Yaskawa INFORM job: A_ROOF_UPPER_0614_2_PAINT_24.JBI

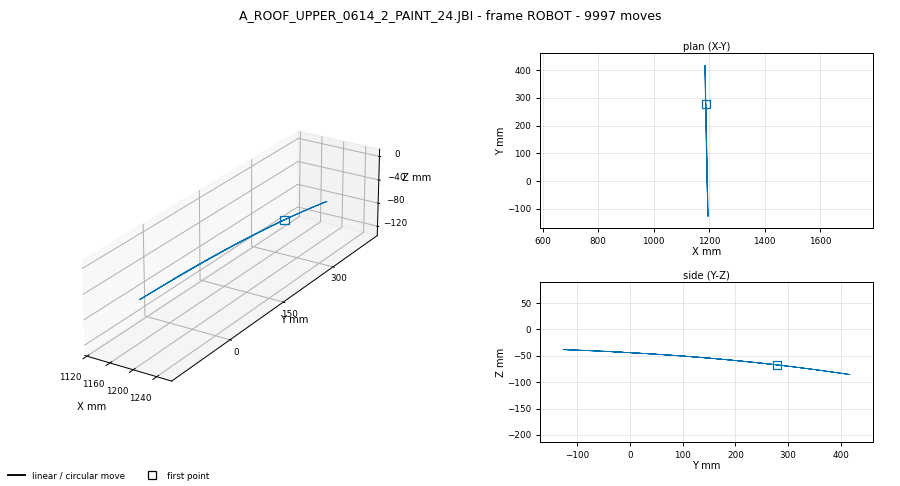
[picture p0: tool path of A_ROOF_UPPER_0614_2_PAINT_24.JBI in frame ROBOT, 9997 of 9997 moves have a stored position in this frame; points joined in program order, loops and branches not executed]
/JOB
//NAME A_ROOF_UPPER_0614_2_PAINT24
//POS
///NPOS 9997,0,0,0,0,0
///TOOL 1
///USER 0
///POSTYPE ROBOT
///RECTAN
///RCONF 1,0,0,0,0,0,0,0,0,0,0,0,0,0,0,0,0,0,0,0,0,0,0,0
C00000=1188.616,279.548,-67.285,-176.910,7.365,148.491
C00001=1188.621,279.299,-67.256,-176.912,7.362,148.491
C00002=1188.625,279.052,-67.228,-176.914,7.359,148.491
C00003=1188.629,278.803,-67.199,-176.917,7.356,148.491
C00004=1188.633,278.555,-67.170,-176.920,7.353,148.491
C00005=1188.638,278.306,-67.142,-176.922,7.351,148.492
C00006=1188.642,278.058,-67.113,-176.925,7.348,148.492
C00007=1188.646,277.809,-67.085,-176.927,7.345,148.492
C00008=1188.651,277.561,-67.056,-176.930,7.343,148.492
C00009=1188.655,277.313,-67.028,-176.932,7.340,148.492
C00010=1188.660,277.065,-67.000,-176.936,7.337,148.492
C00011=1188.664,276.816,-66.971,-176.938,7.335,148.492
C00012=1188.668,276.568,-66.942,-176.940,7.332,148.492
C00013=1188.673,276.320,-66.914,-176.943,7.330,148.492
C00014=1188.677,276.071,-66.885,-176.945,7.327,148.492
C00015=1188.682,275.823,-66.857,-176.948,7.324,148.492
C00016=1188.685,275.574,-66.829,-176.950,7.322,148.492
C00017=1188.690,275.325,-66.800,-176.953,7.319,148.492
C00018=1188.694,275.078,-66.772,-176.956,7.316,148.493
C00019=1188.698,274.829,-66.743,-176.958,7.314,148.493
C00020=1188.703,274.581,-66.715,-176.961,7.311,148.493
C00021=1188.707,274.333,-66.686,-176.964,7.308,148.493
C00022=1188.712,274.085,-66.659,-176.966,7.306,148.493
C00023=1188.716,273.836,-66.630,-176.969,7.303,148.493
C00024=1188.720,273.588,-66.602,-176.971,7.301,148.493
C00025=1188.725,273.339,-66.573,-176.974,7.298,148.493
C00026=1188.729,273.091,-66.546,-176.977,7.295,148.493
C00027=1188.733,272.843,-66.518,-176.979,7.293,148.493
C00028=1188.738,272.594,-66.489,-176.981,7.290,148.493
C00029=1188.742,272.346,-66.461,-176.984,7.287,148.493
C00030=1188.746,272.097,-66.432,-176.986,7.285,148.494
C00031=1188.751,271.849,-66.404,-176.990,7.282,148.494
C00032=1188.755,271.601,-66.377,-176.992,7.280,148.494
C00033=1188.760,271.352,-66.348,-176.994,7.277,148.494
C00034=1188.764,271.104,-66.320,-176.997,7.274,148.494
C00035=1188.768,270.855,-66.291,-176.999,7.272,148.494
C00036=1188.773,270.608,-66.264,-177.002,7.269,148.494
C00037=1188.776,270.359,-66.236,-177.005,7.267,148.494
C00038=1188.782,270.111,-66.207,-177.007,7.264,148.494
C00039=1188.786,269.862,-66.180,-177.010,7.261,148.494
C00040=1188.790,269.614,-66.152,-177.012,7.259,148.495
C00041=1188.794,269.365,-66.123,-177.015,7.256,148.495
C00042=1188.799,269.117,-66.095,-177.018,7.254,148.495
C00043=1188.803,268.868,-66.067,-177.020,7.251,148.495
C00044=1188.808,268.620,-66.039,-177.023,7.248,148.495
C00045=1188.812,268.372,-66.012,-177.025,7.246,148.495
C00046=1188.816,268.123,-65.984,-177.028,7.243,148.495
C00047=1188.821,267.875,-65.955,-177.031,7.241,148.495
C00048=1188.825,267.626,-65.927,-177.033,7.238,148.495
C00049=1188.830,267.378,-65.900,-177.035,7.236,148.496
C00050=1188.834,267.130,-65.872,-177.038,7.233,148.496
C00051=1188.838,266.881,-65.844,-177.041,7.230,148.496
C00052=1188.843,266.633,-65.816,-177.043,7.228,148.496
C00053=1188.847,266.384,-65.788,-177.046,7.225,148.496
C00054=1188.851,266.136,-65.761,-177.048,7.223,148.496
C00055=1188.856,265.888,-65.733,-177.051,7.220,148.496
C00056=1188.860,265.639,-65.705,-177.054,7.218,148.496
C00057=1188.865,265.391,-65.677,-177.056,7.215,148.496
C00058=1188.869,265.143,-65.649,-177.059,7.212,148.497
C00059=1188.873,264.894,-65.622,-177.061,7.210,148.497
C00060=1188.877,264.646,-65.594,-177.064,7.207,148.497
C00061=1188.882,264.396,-65.566,-177.067,7.205,148.497
C00062=1188.887,264.149,-65.538,-177.069,7.202,148.497
C00063=1188.891,263.901,-65.511,-177.072,7.200,148.497
C00064=1188.895,263.652,-65.483,-177.075,7.197,148.497
C00065=1188.899,263.404,-65.455,-177.077,7.194,148.497
C00066=1188.904,263.155,-65.428,-177.080,7.192,148.498
C00067=1188.909,262.882,-65.398,-177.082,7.189,148.498
C00068=1188.914,262.609,-65.367,-177.086,7.186,148.498
C00069=1188.919,262.336,-65.337,-177.088,7.183,148.498
C00070=1188.923,262.064,-65.307,-177.091,7.181,148.498
C00071=1188.928,261.815,-65.280,-177.094,7.179,148.498
C00072=1188.931,261.567,-65.252,-177.096,7.176,148.498
C00073=1188.937,261.318,-65.224,-177.098,7.174,148.498
C00074=1188.941,261.070,-65.196,-177.102,7.171,148.499
C00075=1188.946,260.821,-65.169,-177.104,7.169,148.499
C00076=1188.950,260.573,-65.141,-177.107,7.166,148.499
C00077=1188.954,260.324,-65.114,-177.109,7.164,148.499
C00078=1188.959,260.076,-65.087,-177.112,7.161,148.499
C00079=1188.963,259.827,-65.059,-177.114,7.159,148.499
C00080=1188.967,259.579,-65.032,-177.117,7.156,148.499
C00081=1188.972,259.330,-65.005,-177.120,7.153,148.500
C00082=1188.976,259.082,-64.977,-177.122,7.151,148.500
C00083=1188.980,258.833,-64.949,-177.125,7.148,148.500
C00084=1188.985,258.585,-64.922,-177.128,7.146,148.500
C00085=1188.989,258.337,-64.895,-177.130,7.143,148.500
C00086=1188.994,258.088,-64.868,-177.132,7.141,148.500
C00087=1188.999,257.840,-64.840,-177.135,7.138,148.500
C00088=1189.002,257.592,-64.813,-177.138,7.136,148.500
C00089=1189.006,257.343,-64.786,-177.140,7.133,148.501
C00090=1189.011,257.095,-64.759,-177.143,7.131,148.501
C00091=1189.016,256.846,-64.732,-177.146,7.128,148.501
C00092=1189.020,256.598,-64.705,-177.148,7.126,148.501
C00093=1189.024,256.349,-64.677,-177.151,7.123,148.501
C00094=1189.029,256.100,-64.649,-177.153,7.121,148.501
C00095=1189.033,255.852,-64.622,-177.156,7.118,148.501
C00096=1189.038,255.603,-64.595,-177.158,7.116,148.501
C00097=1189.043,255.355,-64.568,-177.161,7.113,148.502
C00098=1189.046,255.106,-64.541,-177.164,7.111,148.502
C00099=1189.050,254.858,-64.514,-177.166,7.108,148.502
C00100=1189.055,254.610,-64.487,-177.169,7.107,148.502
C00101=1189.060,254.361,-64.460,-177.172,7.104,148.502
C00102=1189.064,254.113,-64.432,-177.174,7.101,148.502
C00103=1189.069,253.864,-64.405,-177.177,7.099,148.503
C00104=1189.073,253.616,-64.379,-177.179,7.097,148.503
C00105=1189.077,253.367,-64.352,-177.182,7.094,148.503
C00106=1189.082,253.118,-64.324,-177.185,7.092,148.503
C00107=1189.086,252.870,-64.297,-177.187,7.089,148.503
C00108=1189.091,252.621,-64.270,-177.189,7.087,148.503
C00109=1189.095,252.373,-64.244,-177.193,7.084,148.504
C00110=1189.100,252.125,-64.217,-177.195,7.082,148.504
C00111=1189.104,251.876,-64.190,-177.197,7.080,148.504
C00112=1189.109,251.628,-64.163,-177.200,7.077,148.504
C00113=1189.113,251.379,-64.136,-177.202,7.075,148.504
C00114=1189.117,251.130,-64.109,-177.206,7.072,148.504
C00115=1189.122,250.882,-64.082,-177.208,7.070,148.504
C00116=1189.126,250.633,-64.055,-177.210,7.067,148.504
C00117=1189.130,250.385,-64.028,-177.213,7.065,148.505
C00118=1189.135,250.137,-64.001,-177.216,7.062,148.505
C00119=1189.140,249.888,-63.975,-177.218,7.060,148.505
C00120=1189.144,249.639,-63.948,-177.221,7.057,148.505
C00121=1189.148,249.391,-63.921,-177.223,7.055,148.505
C00122=1189.153,249.142,-63.894,-177.227,7.053,148.506
C00123=1189.157,248.894,-63.868,-177.229,7.050,148.506
C00124=1189.162,248.646,-63.841,-177.231,7.048,148.506
C00125=1189.166,248.397,-63.814,-177.234,7.046,148.506
C00126=1189.170,248.148,-63.788,-177.236,7.043,148.506
C00127=1189.175,247.900,-63.761,-177.239,7.041,148.506
C00128=1189.180,247.651,-63.734,-177.242,7.039,148.507
C00129=1189.184,247.403,-63.707,-177.245,7.036,148.507
C00130=1189.189,247.154,-63.681,-177.247,7.034,148.507
C00131=1189.193,246.906,-63.654,-177.250,7.031,148.507
C00132=1189.197,246.657,-63.627,-177.252,7.029,148.507
C00133=1189.202,246.409,-63.600,-177.255,7.027,148.507
C00134=1189.206,246.160,-63.575,-177.258,7.024,148.508
C00135=1189.211,245.912,-63.548,-177.260,7.022,148.508
C00136=1189.215,245.663,-63.521,-177.263,7.019,148.508
C00137=1189.220,245.414,-63.495,-177.265,7.017,148.508
C00138=1189.224,245.166,-63.468,-177.268,7.014,148.508
C00139=1189.228,244.918,-63.441,-177.271,7.012,148.509
C00140=1189.232,244.669,-63.415,-177.273,7.010,148.509
C00141=1189.237,244.420,-63.388,-177.276,7.008,148.509
C00142=1189.241,244.171,-63.363,-177.278,7.005,148.509
C00143=1189.246,243.923,-63.336,-177.281,7.002,148.509
C00144=1189.250,243.675,-63.309,-177.284,7.001,148.509
C00145=1189.255,243.426,-63.283,-177.286,6.998,148.509
C00146=1189.259,243.178,-63.256,-177.289,6.996,148.510
C00147=1189.264,242.928,-63.230,-177.291,6.994,148.510
C00148=1189.268,242.680,-63.203,-177.294,6.991,148.510
C00149=1189.273,242.431,-63.177,-177.296,6.989,148.510
C00150=1189.277,242.184,-63.151,-177.299,6.987,148.511
C00151=1189.282,241.935,-63.125,-177.302,6.984,148.511
C00152=1189.286,241.686,-63.098,-177.304,6.982,148.511
C00153=1189.291,241.437,-63.072,-177.307,6.979,148.511
C00154=1189.295,241.189,-63.045,-177.310,6.977,148.511
C00155=1189.299,240.940,-63.020,-177.312,6.975,148.511
C00156=1189.304,240.692,-62.993,-177.315,6.972,148.511
C00157=1189.308,240.443,-62.967,-177.317,6.970,148.512
C00158=1189.313,240.194,-62.941,-177.320,6.967,148.512
C00159=1189.317,239.946,-62.914,-177.323,6.966,148.512
C00160=1189.322,239.698,-62.889,-177.325,6.963,148.512
C00161=1189.326,239.449,-62.862,-177.328,6.961,148.513
C00162=1189.331,239.200,-62.836,-177.330,6.959,148.513
C00163=1189.335,238.951,-62.810,-177.333,6.956,148.513
C00164=1189.339,238.703,-62.783,-177.336,6.954,148.513
C00165=1189.344,238.454,-62.757,-177.338,6.952,148.513
C00166=1189.348,238.206,-62.732,-177.341,6.949,148.513
C00167=1189.353,237.958,-62.705,-177.344,6.947,148.514
C00168=1189.357,237.709,-62.679,-177.346,6.945,148.514
C00169=1189.362,237.460,-62.653,-177.349,6.942,148.514
C00170=1189.367,237.211,-62.627,-177.351,6.940,148.514
C00171=1189.372,236.940,-62.599,-177.354,6.938,148.515
C00172=1189.376,236.668,-62.571,-177.358,6.935,148.515
C00173=1189.381,236.397,-62.542,-177.360,6.933,148.515
C00174=1189.385,236.125,-62.514,-177.363,6.930,148.515
C00175=1189.391,235.877,-62.488,-177.366,6.928,148.516
C00176=1189.395,235.629,-62.461,-177.368,6.925,148.516
C00177=1189.399,235.380,-62.436,-177.371,6.923,148.516
C00178=1189.403,235.131,-62.410,-177.373,6.921,148.516
C00179=1189.408,234.882,-62.383,-177.376,6.919,148.516
C00180=1189.413,234.634,-62.358,-177.379,6.916,148.516
C00181=1189.417,234.385,-62.332,-177.381,6.915,148.517
C00182=1189.421,234.136,-62.307,-177.384,6.912,148.517
C00183=1189.425,233.888,-62.280,-177.387,6.910,148.517
C00184=1189.431,233.639,-62.254,-177.389,6.908,148.517
C00185=1189.435,233.391,-62.228,-177.392,6.905,148.518
C00186=1189.439,233.142,-62.203,-177.394,6.903,148.518
C00187=1189.444,232.893,-62.177,-177.397,6.901,148.518
C00188=1189.448,232.645,-62.151,-177.400,6.898,148.518
C00189=1189.453,232.396,-62.126,-177.402,6.896,148.518
C00190=1189.457,232.147,-62.100,-177.405,6.894,148.519
C00191=1189.462,231.899,-62.074,-177.407,6.891,148.519
C00192=1189.467,231.650,-62.048,-177.410,6.890,148.519
C00193=1189.471,231.401,-62.023,-177.412,6.887,148.519
C00194=1189.475,231.153,-61.997,-177.416,6.885,148.519
C00195=1189.480,230.904,-61.971,-177.418,6.883,148.520
C00196=1189.484,230.656,-61.946,-177.420,6.881,148.520
C00197=1189.488,230.407,-61.920,-177.424,6.878,148.520
C00198=1189.493,230.159,-61.894,-177.426,6.876,148.520
C00199=1189.497,229.910,-61.869,-177.428,6.874,148.521
C00200=1189.502,229.661,-61.843,-177.431,6.871,148.521
C00201=1189.507,229.412,-61.818,-177.434,6.869,148.521
C00202=1189.511,229.164,-61.793,-177.436,6.868,148.521
C00203=1189.515,228.915,-61.767,-177.439,6.865,148.521
C00204=1189.520,228.667,-61.741,-177.442,6.863,148.522
C00205=1189.524,228.418,-61.716,-177.444,6.861,148.522
C00206=1189.529,228.169,-61.690,-177.447,6.858,148.522
C00207=1189.533,227.921,-61.665,-177.450,6.856,148.522
C00208=1189.538,227.672,-61.640,-177.452,6.854,148.523
C00209=1189.543,227.423,-61.614,-177.455,6.852,148.523
C00210=1189.547,227.175,-61.588,-177.457,6.849,148.523
C00211=1189.551,226.926,-61.563,-177.460,6.847,148.523
C00212=1189.556,226.678,-61.537,-177.463,6.846,148.524
C00213=1189.561,226.428,-61.512,-177.465,6.843,148.524
C00214=1189.565,226.179,-61.486,-177.468,6.841,148.524
C00215=1189.570,225.931,-61.461,-177.471,6.839,148.524
C00216=1189.574,225.682,-61.436,-177.473,6.836,148.524
C00217=1189.579,225.434,-61.411,-177.476,6.834,148.525
C00218=1189.583,225.185,-61.385,-177.478,6.832,148.525
C00219=1189.588,224.937,-61.360,-177.481,6.830,148.525
C00220=1189.593,224.688,-61.334,-177.484,6.828,148.526
C00221=1189.597,224.439,-61.309,-177.486,6.825,148.526
C00222=1189.602,224.190,-61.284,-177.489,6.824,148.526
C00223=1189.605,223.941,-61.259,-177.492,6.821,148.526
C00224=1189.610,223.693,-61.234,-177.494,6.819,148.526
C00225=1189.615,223.444,-61.208,-177.497,6.817,148.527
C00226=1189.620,223.196,-61.183,-177.500,6.815,148.527
C00227=1189.624,222.947,-61.157,-177.502,6.812,148.527
C00228=1189.629,222.698,-61.133,-177.505,6.810,148.527
C00229=1189.632,222.450,-61.108,-177.507,6.808,148.528
C00230=1189.638,222.201,-61.083,-177.510,6.806,148.528
C00231=1189.642,221.952,-61.057,-177.513,6.804,148.528
C00232=1189.646,221.703,-61.032,-177.515,6.802,148.528
C00233=1189.651,221.455,-61.007,-177.518,6.800,148.529
C00234=1189.655,221.206,-60.982,-177.521,6.797,148.529
C00235=1189.660,220.958,-60.957,-177.523,6.795,148.529
C00236=1189.664,220.708,-60.932,-177.526,6.793,148.529
C00237=1189.669,220.460,-60.906,-177.529,6.791,148.530
C00238=1189.674,220.211,-60.881,-177.531,6.788,148.530
C00239=1189.678,219.963,-60.857,-177.534,6.787,148.530
C00240=1189.682,219.713,-60.832,-177.537,6.785,148.530
C00241=1189.687,219.465,-60.806,-177.539,6.783,148.531
C00242=1189.691,219.217,-60.782,-177.542,6.780,148.531
C00243=1189.696,218.967,-60.757,-177.545,6.778,148.531
C00244=1189.701,218.719,-60.732,-177.547,6.776,148.532
C00245=1189.705,218.470,-60.707,-177.549,6.774,148.532
C00246=1189.709,218.222,-60.682,-177.553,6.772,148.532
C00247=1189.714,217.973,-60.657,-177.555,6.770,148.532
C00248=1189.719,217.724,-60.632,-177.557,6.768,148.532
C00249=1189.723,217.475,-60.607,-177.560,6.766,148.533
C00250=1189.728,217.227,-60.582,-177.563,6.763,148.533
C00251=1189.733,216.978,-60.558,-177.565,6.761,148.533
C00252=1189.737,216.729,-60.533,-177.568,6.759,148.533
C00253=1189.741,216.481,-60.508,-177.571,6.757,148.534
C00254=1189.745,216.232,-60.483,-177.574,6.755,148.534
C00255=1189.750,215.983,-60.459,-177.576,6.753,148.534
C00256=1189.755,215.734,-60.433,-177.579,6.751,148.535
C00257=1189.759,215.486,-60.409,-177.581,6.749,148.535
C00258=1189.764,215.237,-60.384,-177.584,6.747,148.535
C00259=1189.769,214.988,-60.359,-177.587,6.744,148.535
C00260=1189.773,214.739,-60.335,-177.590,6.742,148.536
C00261=1189.778,214.491,-60.310,-177.592,6.741,148.536
C00262=1189.782,214.242,-60.285,-177.594,6.738,148.536
C00263=1189.787,213.993,-60.261,-177.598,6.736,148.536
C00264=1189.791,213.744,-60.236,-177.600,6.734,148.537
C00265=1189.796,213.495,-60.212,-177.603,6.732,148.537
C00266=1189.800,213.247,-60.187,-177.605,6.730,148.537
C00267=1189.804,212.998,-60.162,-177.608,6.727,148.537
C00268=1189.809,212.750,-60.138,-177.611,6.726,148.538
C00269=1189.814,212.501,-60.113,-177.613,6.723,148.538
C00270=1189.818,212.252,-60.088,-177.616,6.722,148.538
C00271=1189.823,212.003,-60.064,-177.618,6.720,148.539
C00272=1189.828,211.755,-60.039,-177.622,6.717,148.539
C00273=1189.832,211.505,-60.015,-177.624,6.715,148.539
C00274=1189.836,211.257,-59.991,-177.626,6.713,148.539
C00275=1189.841,210.987,-59.964,-177.629,6.711,148.540
C00276=1189.846,210.717,-59.937,-177.632,6.709,148.540
C00277=1189.851,210.446,-59.910,-177.635,6.707,148.540
C00278=1189.856,210.175,-59.884,-177.638,6.704,148.541
C00279=1189.861,209.927,-59.860,-177.641,6.703,148.541
C00280=1189.865,209.677,-59.835,-177.643,6.700,148.541
C00281=1189.870,209.429,-59.811,-177.646,6.699,148.541
C00282=1189.875,209.180,-59.786,-177.649,6.696,148.542
C00283=1189.879,208.932,-59.762,-177.652,6.694,148.542
C00284=1189.883,208.682,-59.738,-177.654,6.692,148.542
C00285=1189.888,208.434,-59.713,-177.656,6.690,148.543
C00286=1189.893,208.185,-59.689,-177.659,6.688,148.543
C00287=1189.898,207.937,-59.664,-177.662,6.686,148.543
C00288=1189.902,207.688,-59.640,-177.664,6.684,148.543
C00289=1189.906,207.438,-59.617,-177.667,6.682,148.544
C00290=1189.911,207.190,-59.592,-177.670,6.680,148.544
C00291=1189.916,206.941,-59.568,-177.672,6.678,148.544
C00292=1189.920,206.692,-59.543,-177.676,6.676,148.545
C00293=1189.925,206.444,-59.519,-177.678,6.673,148.545
C00294=1189.929,206.195,-59.495,-177.681,6.672,148.545
C00295=1189.934,205.946,-59.471,-177.683,6.670,148.545
C00296=1189.939,205.697,-59.447,-177.686,6.668,148.546
C00297=1189.943,205.448,-59.422,-177.688,6.666,148.546
C00298=1189.947,205.200,-59.398,-177.691,6.663,148.546
C00299=1189.953,204.950,-59.374,-177.694,6.661,148.547
C00300=1189.957,204.702,-59.350,-177.697,6.660,148.547
C00301=1189.961,204.454,-59.326,-177.699,6.658,148.547
C00302=1189.965,204.205,-59.302,-177.702,6.656,148.548
C00303=1189.971,203.955,-59.278,-177.704,6.654,148.548
C00304=1189.975,203.707,-59.254,-177.707,6.652,148.548
C00305=1189.979,203.458,-59.229,-177.710,6.649,148.548
C00306=1189.984,203.209,-59.206,-177.713,6.648,148.549
C00307=1189.989,202.961,-59.181,-177.715,6.646,148.549
C00308=1189.993,202.712,-59.157,-177.717,6.644,148.549
C00309=1189.998,202.462,-59.134,-177.720,6.642,148.550
C00310=1190.002,202.214,-59.110,-177.723,6.640,148.550
C00311=1190.006,201.966,-59.085,-177.725,6.638,148.550
C00312=1190.011,201.717,-59.062,-177.729,6.636,148.551
C00313=1190.016,201.468,-59.037,-177.731,6.633,148.551
C00314=1190.021,201.219,-59.014,-177.733,6.632,148.551
C00315=1190.025,200.970,-58.990,-177.736,6.630,148.551
C00316=1190.029,200.721,-58.966,-177.739,6.628,148.552
C00317=1190.034,200.472,-58.942,-177.741,6.626,148.552
C00318=1190.038,200.224,-58.918,-177.744,6.624,148.552
C00319=1190.044,199.975,-58.894,-177.747,6.621,148.553
C00320=1190.048,199.726,-58.870,-177.749,6.620,148.553
C00321=1190.053,199.477,-58.847,-177.752,6.618,148.553
C00322=1190.057,199.229,-58.823,-177.755,6.616,148.554
C00323=1190.062,198.980,-58.799,-177.757,6.614,148.554
C00324=1190.067,198.731,-58.776,-177.760,6.612,148.554
C00325=1190.071,198.482,-58.752,-177.762,6.610,148.554
C00326=1190.076,198.233,-58.729,-177.765,6.608,148.555
C00327=1190.079,197.984,-58.704,-177.768,6.606,148.555
C00328=1190.084,197.735,-58.681,-177.771,6.604,148.555
C00329=1190.089,197.487,-58.657,-177.774,6.602,148.556
C00330=1190.093,197.238,-58.633,-177.776,6.600,148.556
C00331=1190.098,196.989,-58.610,-177.778,6.598,148.556
C00332=1190.103,196.740,-58.585,-177.781,6.597,148.557
C00333=1190.108,196.491,-58.562,-177.784,6.595,148.557
C00334=1190.113,196.242,-58.539,-177.786,6.593,148.557
C00335=1190.117,195.993,-58.514,-177.789,6.591,148.558
C00336=1190.122,195.744,-58.491,-177.792,6.589,148.558
C00337=1190.126,195.495,-58.468,-177.795,6.587,148.558
C00338=1190.131,195.247,-58.444,-177.797,6.585,148.558
C00339=1190.135,194.998,-58.420,-177.800,6.583,148.559
C00340=1190.140,194.749,-58.397,-177.802,6.581,148.559
C00341=1190.144,194.501,-58.373,-177.805,6.579,148.559
C00342=1190.148,194.252,-58.350,-177.808,6.577,148.560
C00343=1190.153,194.003,-58.327,-177.810,6.576,148.560
C00344=1190.158,193.754,-58.303,-177.813,6.574,148.560
C00345=1190.162,193.505,-58.279,-177.816,6.572,148.561
C00346=1190.167,193.256,-58.256,-177.818,6.570,148.561
C00347=1190.172,193.007,-58.233,-177.821,6.568,148.561
C00348=1190.176,192.758,-58.209,-177.824,6.565,148.562
C00349=1190.181,192.509,-58.186,-177.826,6.564,148.562
C00350=1190.185,192.261,-58.162,-177.829,6.562,148.562
C00351=1190.191,192.012,-58.139,-177.832,6.560,148.563
C00352=1190.195,191.763,-58.115,-177.834,6.558,148.563
C00353=1190.199,191.515,-58.093,-177.837,6.556,148.563
C00354=1190.204,191.266,-58.069,-177.840,6.555,148.564
C00355=1190.209,191.017,-58.046,-177.842,6.552,148.564
C00356=1190.213,190.767,-58.023,-177.845,6.551,148.564
C00357=1190.218,190.518,-57.999,-177.847,6.549,148.565
C00358=1190.223,190.269,-57.976,-177.850,6.547,148.565
C00359=1190.227,190.021,-57.952,-177.853,6.545,148.565
C00360=1190.231,189.772,-57.929,-177.855,6.543,148.566
C00361=1190.236,189.523,-57.906,-177.858,6.542,148.566
C00362=1190.241,189.274,-57.882,-177.861,6.540,148.566
C00363=1190.246,189.026,-57.859,-177.864,6.537,148.567
C00364=1190.251,188.777,-57.836,-177.866,6.535,148.567
C00365=1190.255,188.528,-57.813,-177.869,6.533,148.567
C00366=1190.259,188.279,-57.790,-177.871,6.531,148.568
C00367=1190.264,188.030,-57.767,-177.874,6.530,148.568
C00368=1190.269,187.781,-57.743,-177.877,6.528,148.568
C00369=1190.273,187.532,-57.720,-177.879,6.526,148.569
C00370=1190.277,187.283,-57.697,-177.882,6.524,148.569
C00371=1190.283,187.034,-57.675,-177.885,6.523,148.569
C00372=1190.288,186.785,-57.651,-177.887,6.521,148.570
C00373=1190.292,186.537,-57.629,-177.890,6.519,148.570
C00374=1190.296,186.288,-57.605,-177.893,6.517,148.570
C00375=1190.301,186.039,-57.582,-177.895,6.515,148.571
C00376=1190.306,185.789,-57.559,-177.898,6.514,148.571
C00377=1190.310,185.541,-57.536,-177.901,6.512,148.571
C00378=1190.315,185.292,-57.513,-177.903,6.510,148.572
C00379=1190.320,185.023,-57.488,-177.906,6.508,148.572
C00380=1190.325,184.753,-57.463,-177.909,6.506,148.572
C00381=1190.330,184.483,-57.438,-177.912,6.504,148.573
C00382=1190.335,184.214,-57.414,-177.915,6.502,148.573
C00383=1190.340,183.965,-57.391,-177.917,6.500,148.574
C00384=1190.344,183.716,-57.367,-177.920,6.498,148.574
C00385=1190.348,183.467,-57.345,-177.923,6.497,148.574
C00386=1190.354,183.218,-57.322,-177.925,6.495,148.575
C00387=1190.358,182.969,-57.299,-177.928,6.493,148.575
C00388=1190.362,182.721,-57.276,-177.931,6.491,148.575
C00389=1190.367,182.471,-57.253,-177.933,6.489,148.576
C00390=1190.371,182.222,-57.231,-177.935,6.487,148.576
C00391=1190.377,181.974,-57.208,-177.938,6.485,148.576
C00392=1190.381,181.725,-57.185,-177.941,6.484,148.576
C00393=1190.386,181.475,-57.162,-177.943,6.482,148.577
C00394=1190.390,181.226,-57.139,-177.946,6.480,148.577
C00395=1190.395,180.978,-57.116,-177.949,6.478,148.578
C00396=1190.400,180.729,-57.094,-177.951,6.476,148.578
C00397=1190.404,180.480,-57.071,-177.954,6.475,148.578
C00398=1190.409,180.232,-57.048,-177.957,6.473,148.579
C00399=1190.413,179.982,-57.026,-177.959,6.471,148.579
C00400=1190.418,179.733,-57.003,-177.962,6.469,148.579
C00401=1190.422,179.484,-56.981,-177.965,6.468,148.580
C00402=1190.428,179.236,-56.958,-177.967,6.466,148.580
C00403=1190.432,178.987,-56.935,-177.970,6.464,148.580
C00404=1190.437,178.737,-56.912,-177.973,6.462,148.581
C00405=1190.441,178.489,-56.890,-177.975,6.460,148.581
C00406=1190.446,178.240,-56.867,-177.978,6.459,148.582
C00407=1190.450,177.991,-56.844,-177.981,6.457,148.582
C00408=1190.456,177.742,-56.822,-177.983,6.455,148.582
C00409=1190.460,177.493,-56.799,-177.986,6.453,148.583
C00410=1190.465,177.244,-56.777,-177.989,6.451,148.583
C00411=1190.469,176.995,-56.754,-177.991,6.450,148.583
C00412=1190.474,176.746,-56.732,-177.994,6.448,148.584
C00413=1190.478,176.497,-56.709,-177.997,6.446,148.584
C00414=1190.483,176.248,-56.687,-177.999,6.444,148.584
C00415=1190.488,175.999,-56.664,-178.002,6.442,148.585
C00416=1190.492,175.750,-56.642,-178.005,6.441,148.585
C00417=1190.497,175.501,-56.620,-178.008,6.439,148.585
C00418=1190.502,175.252,-56.597,-178.010,6.437,148.586
C00419=1190.506,175.003,-56.575,-178.013,6.435,148.586
C00420=1190.511,174.755,-56.552,-178.016,6.434,148.587
C00421=1190.516,174.505,-56.530,-178.018,6.432,148.587
C00422=1190.520,174.256,-56.508,-178.021,6.430,148.587
C00423=1190.525,174.008,-56.485,-178.024,6.428,148.588
C00424=1190.529,173.758,-56.463,-178.026,6.426,148.588
C00425=1190.534,173.510,-56.441,-178.028,6.425,148.588
C00426=1190.539,173.261,-56.418,-178.031,6.424,148.589
C00427=1190.543,173.011,-56.395,-178.034,6.422,148.589
C00428=1190.548,172.763,-56.374,-178.036,6.420,148.589
C00429=1190.553,172.514,-56.350,-178.039,6.418,148.590
C00430=1190.558,172.265,-56.329,-178.042,6.416,148.590
C00431=1190.562,172.016,-56.307,-178.044,6.415,148.591
C00432=1190.568,171.767,-56.284,-178.047,6.413,148.591
C00433=1190.572,171.518,-56.262,-178.050,6.411,148.591
C00434=1190.576,171.269,-56.240,-178.052,6.409,148.592
C00435=1190.581,171.020,-56.218,-178.055,6.408,148.592
C00436=1190.586,170.770,-56.195,-178.058,6.406,148.592
C00437=1190.590,170.522,-56.173,-178.060,6.404,148.593
C00438=1190.595,170.273,-56.151,-178.063,6.402,148.593
C00439=1190.599,170.024,-56.129,-178.066,6.400,148.593
C00440=1190.604,169.775,-56.107,-178.068,6.399,148.594
C00441=1190.609,169.526,-56.085,-178.071,6.398,148.594
C00442=1190.614,169.277,-56.063,-178.074,6.396,148.595
C00443=1190.618,169.029,-56.040,-178.076,6.394,148.595
C00444=1190.622,168.779,-56.018,-178.079,6.393,148.596
C00445=1190.628,168.531,-55.996,-178.082,6.391,148.596
C00446=1190.632,168.281,-55.974,-178.084,6.389,148.596
C00447=1190.637,168.033,-55.952,-178.087,6.387,148.597
C00448=1190.641,167.783,-55.930,-178.090,6.385,148.597
C00449=1190.646,167.535,-55.909,-178.092,6.384,148.597
C00450=1190.651,167.285,-55.886,-178.095,6.382,148.598
C00451=1190.656,167.036,-55.864,-178.097,6.381,148.598
C00452=1190.660,166.787,-55.842,-178.100,6.379,148.599
C00453=1190.665,166.538,-55.821,-178.103,6.377,148.599
C00454=1190.670,166.289,-55.798,-178.105,6.376,148.599
C00455=1190.674,166.040,-55.777,-178.108,6.374,148.600
C00456=1190.679,165.791,-55.755,-178.111,6.372,148.600
C00457=1190.684,165.542,-55.733,-178.113,6.370,148.600
C00458=1190.688,165.294,-55.711,-178.116,6.368,148.601
C00459=1190.693,165.044,-55.689,-178.119,6.367,148.601
C00460=1190.698,164.795,-55.667,-178.122,6.365,148.602
C00461=1190.703,164.546,-55.645,-178.124,6.364,148.602
C00462=1190.707,164.297,-55.623,-178.127,6.362,148.602
C00463=1190.712,164.048,-55.601,-178.129,6.361,148.603
C00464=1190.717,163.799,-55.580,-178.132,6.359,148.603
C00465=1190.721,163.550,-55.558,-178.135,6.357,148.604
C00466=1190.726,163.301,-55.536,-178.137,6.355,148.604
C00467=1190.731,163.053,-55.514,-178.140,6.354,148.604
C00468=1190.735,162.803,-55.492,-178.143,6.352,148.605
C00469=1190.740,162.554,-55.471,-178.145,6.351,148.605
C00470=1190.744,162.305,-55.449,-178.147,6.349,148.605
C00471=1190.749,162.056,-55.427,-178.151,6.348,148.606
C00472=1190.754,161.808,-55.406,-178.153,6.346,148.606
C00473=1190.758,161.558,-55.384,-178.156,6.344,148.607
C00474=1190.763,161.310,-55.362,-178.159,6.342,148.607
C00475=1190.768,161.060,-55.341,-178.161,6.341,148.607
C00476=1190.773,160.811,-55.319,-178.163,6.340,148.608
C00477=1190.777,160.562,-55.297,-178.166,6.338,148.608
C00478=1190.782,160.313,-55.275,-178.169,6.336,148.609
C00479=1190.787,160.064,-55.254,-178.171,6.334,148.609
C00480=1190.792,159.815,-55.233,-178.174,6.332,148.609
C00481=1190.795,159.566,-55.211,-178.177,6.331,148.610
C00482=1190.800,159.317,-55.190,-178.180,6.329,148.610
C00483=1190.806,159.048,-55.166,-178.183,6.327,148.611
C00484=1190.810,158.779,-55.143,-178.185,6.326,148.611
C00485=1190.816,158.510,-55.119,-178.188,6.324,148.612
C00486=1190.820,158.241,-55.097,-178.191,6.322,148.612
C00487=1190.825,157.992,-55.076,-178.194,6.321,148.612
C00488=1190.830,157.743,-55.054,-178.196,6.319,148.613
C00489=1190.835,157.494,-55.032,-178.199,6.318,148.613
C00490=1190.840,157.245,-55.011,-178.201,6.316,148.614
C00491=1190.845,156.996,-54.989,-178.204,6.314,148.614
C00492=1190.850,156.747,-54.968,-178.207,6.313,148.615
C00493=1190.853,156.498,-54.947,-178.210,6.311,148.615
C00494=1190.858,156.249,-54.925,-178.212,6.309,148.615
C00495=1190.863,156.000,-54.904,-178.215,6.308,148.616
C00496=1190.868,155.751,-54.882,-178.217,6.307,148.616
C00497=1190.873,155.502,-54.860,-178.220,6.305,148.616
C00498=1190.878,155.253,-54.839,-178.223,6.303,148.617
C00499=1190.882,155.004,-54.818,-178.226,6.302,148.617
C00500=1190.886,154.754,-54.797,-178.228,6.300,148.618
C00501=1190.891,154.506,-54.775,-178.231,6.299,148.618
C00502=1190.896,154.256,-54.754,-178.233,6.297,148.619
C00503=1190.901,154.008,-54.733,-178.236,6.295,148.619
C00504=1190.905,153.758,-54.712,-178.239,6.294,148.619
C00505=1190.910,153.510,-54.690,-178.241,6.292,148.620
C00506=1190.915,153.260,-54.669,-178.244,6.291,148.620
C00507=1190.920,153.011,-54.649,-178.247,6.289,148.621
C00508=1190.925,152.763,-54.627,-178.249,6.288,148.621
C00509=1190.929,152.513,-54.606,-178.252,6.286,148.621
C00510=1190.934,152.264,-54.584,-178.255,6.284,148.622
C00511=1190.938,152.015,-54.564,-178.257,6.283,148.622
C00512=1190.943,151.767,-54.542,-178.260,6.282,148.623
C00513=1190.948,151.517,-54.521,-178.263,6.280,148.623
C00514=1190.952,151.268,-54.500,-178.265,6.278,148.624
C00515=1190.957,151.019,-54.479,-178.268,6.276,148.624
C00516=1190.962,150.770,-54.458,-178.270,6.275,148.624
C00517=1190.968,150.520,-54.437,-178.273,6.274,148.625
C00518=1190.972,150.272,-54.416,-178.276,6.272,148.625
C00519=1190.976,150.022,-54.394,-178.279,6.271,148.626
C00520=1190.981,149.773,-54.374,-178.281,6.269,148.626
C00521=1190.986,149.525,-54.352,-178.283,6.268,148.626
C00522=1190.991,149.275,-54.331,-178.286,6.266,148.627
C00523=1190.995,149.026,-54.311,-178.289,6.264,148.627
C00524=1191.000,148.778,-54.289,-178.292,6.263,148.628
C00525=1191.005,148.528,-54.268,-178.295,6.261,148.628
C00526=1191.009,148.279,-54.248,-178.297,6.260,148.629
C00527=1191.014,148.030,-54.227,-178.299,6.258,148.629
C00528=1191.018,147.781,-54.206,-178.302,6.257,148.629
C00529=1191.023,147.532,-54.185,-178.305,6.255,148.630
C00530=1191.029,147.283,-54.164,-178.307,6.254,148.630
C00531=1191.033,147.034,-54.143,-178.310,6.252,148.631
C00532=1191.038,146.784,-54.122,-178.313,6.251,148.631
C00533=1191.042,146.536,-54.101,-178.315,6.249,148.631
C00534=1191.048,146.287,-54.080,-178.318,6.248,148.632
C00535=1191.051,146.037,-54.060,-178.321,6.246,148.632
C00536=1191.057,145.788,-54.039,-178.323,6.245,148.633
C00537=1191.061,145.539,-54.018,-178.326,6.243,148.633
C00538=1191.066,145.290,-53.997,-178.328,6.242,148.634
C00539=1191.071,145.041,-53.977,-178.331,6.240,148.634
C00540=1191.076,144.792,-53.956,-178.334,6.239,148.635
C00541=1191.080,144.543,-53.935,-178.337,6.237,148.635
C00542=1191.085,144.294,-53.914,-178.339,6.236,148.635
C00543=1191.090,144.045,-53.893,-178.342,6.234,148.636
C00544=1191.095,143.796,-53.872,-178.344,6.233,148.636
C00545=1191.099,143.547,-53.852,-178.347,6.231,148.637
C00546=1191.104,143.298,-53.831,-178.350,6.230,148.637
C00547=1191.109,143.049,-53.811,-178.352,6.228,148.638
C00548=1191.114,142.799,-53.790,-178.355,6.227,148.638
C00549=1191.118,142.550,-53.769,-178.358,6.225,148.639
C00550=1191.122,142.301,-53.749,-178.360,6.224,148.639
C00551=1191.127,142.051,-53.728,-178.363,6.222,148.639
C00552=1191.132,141.803,-53.707,-178.366,6.221,148.640
C00553=1191.137,141.553,-53.686,-178.368,6.219,148.640
C00554=1191.141,141.304,-53.666,-178.371,6.218,148.641
C00555=1191.146,141.055,-53.646,-178.374,6.217,148.641
C00556=1191.151,140.806,-53.625,-178.376,6.215,148.642
C00557=1191.156,140.557,-53.604,-178.379,6.213,148.642
C00558=1191.161,140.308,-53.583,-178.381,6.212,148.643
C00559=1191.165,140.059,-53.563,-178.384,6.211,148.643
C00560=1191.170,139.809,-53.543,-178.387,6.209,148.643
C00561=1191.175,139.560,-53.522,-178.389,6.208,148.644
C00562=1191.179,139.311,-53.502,-178.392,6.207,148.644
C00563=1191.184,139.062,-53.482,-178.395,6.205,148.645
C00564=1191.189,138.813,-53.461,-178.398,6.203,148.645
C00565=1191.194,138.565,-53.441,-178.400,6.202,148.645
C00566=1191.199,138.316,-53.420,-178.403,6.201,148.646
C00567=1191.204,138.066,-53.400,-178.406,6.199,148.646
C00568=1191.208,137.817,-53.380,-178.408,6.198,148.647
C00569=1191.213,137.568,-53.359,-178.410,6.196,148.647
C00570=1191.218,137.319,-53.338,-178.413,6.195,148.648
C00571=1191.223,137.070,-53.318,-178.416,6.193,148.648
C00572=1191.227,136.820,-53.298,-178.418,6.192,148.649
C00573=1191.232,136.571,-53.278,-178.421,6.190,148.649
C00574=1191.237,136.322,-53.257,-178.424,6.189,148.650
C00575=1191.241,136.073,-53.237,-178.426,6.188,148.650
C00576=1191.246,135.823,-53.217,-178.429,6.186,148.650
C00577=1191.251,135.575,-53.197,-178.432,6.184,148.651
C00578=1191.256,135.325,-53.176,-178.434,6.184,148.651
C00579=1191.261,135.077,-53.156,-178.437,6.182,148.652
C00580=1191.265,134.827,-53.136,-178.440,6.180,148.652
C00581=1191.270,134.579,-53.116,-178.442,6.179,148.653
C00582=1191.275,134.329,-53.095,-178.445,6.178,148.653
C00583=1191.280,134.080,-53.075,-178.448,6.176,148.654
C00584=1191.284,133.831,-53.055,-178.450,6.175,148.654
C00585=1191.289,133.582,-53.034,-178.452,6.173,148.654
C00586=1191.293,133.332,-53.015,-178.456,6.172,148.655
C00587=1191.299,133.064,-52.992,-178.458,6.170,148.655
C00588=1191.304,132.795,-52.971,-178.461,6.169,148.656
C00589=1191.309,132.526,-52.949,-178.464,6.168,148.656
C00590=1191.314,132.258,-52.928,-178.467,6.167,148.657
C00591=1191.319,132.008,-52.907,-178.469,6.165,148.657
C00592=1191.324,131.759,-52.887,-178.472,6.163,148.658
C00593=1191.329,131.511,-52.868,-178.474,6.162,148.658
C00594=1191.334,131.262,-52.847,-178.477,6.161,148.659
C00595=1191.338,131.013,-52.827,-178.480,6.159,148.659
C00596=1191.343,130.763,-52.807,-178.482,6.158,148.660
C00597=1191.347,130.514,-52.787,-178.485,6.157,148.660
C00598=1191.353,130.265,-52.768,-178.488,6.155,148.661
C00599=1191.357,130.016,-52.747,-178.490,6.154,148.661
C00600=1191.363,129.766,-52.727,-178.493,6.152,148.661
C00601=1191.367,129.517,-52.707,-178.496,6.151,148.662
C00602=1191.372,129.268,-52.687,-178.498,6.150,148.662
C00603=1191.377,129.019,-52.668,-178.501,6.148,148.663
C00604=1191.381,128.770,-52.647,-178.504,6.147,148.663
C00605=1191.386,128.521,-52.628,-178.506,6.146,148.664
C00606=1191.391,128.272,-52.607,-178.509,6.144,148.664
C00607=1191.395,128.022,-52.588,-178.512,6.142,148.665
C00608=1191.400,127.774,-52.568,-178.514,6.142,148.665
C00609=1191.405,127.524,-52.548,-178.517,6.140,148.666
C00610=1191.410,127.275,-52.528,-178.520,6.139,148.666
C00611=1191.414,127.026,-52.508,-178.522,6.137,148.667
C00612=1191.420,126.777,-52.489,-178.525,6.136,148.667
C00613=1191.424,126.527,-52.469,-178.527,6.135,148.668
C00614=1191.429,126.278,-52.449,-178.530,6.133,148.668
C00615=1191.434,126.029,-52.429,-178.533,6.132,148.669
C00616=1191.439,125.780,-52.410,-178.535,6.131,148.669
C00617=1191.443,125.531,-52.389,-178.538,6.129,148.670
C00618=1191.448,125.281,-52.370,-178.540,6.128,148.670
C00619=1191.453,125.032,-52.350,-178.543,6.127,148.670
C00620=1191.458,124.784,-52.330,-178.546,6.125,148.671
C00621=1191.463,124.534,-52.310,-178.548,6.124,148.671
C00622=1191.467,124.285,-52.291,-178.551,6.122,148.672
C00623=1191.472,124.036,-52.272,-178.554,6.121,148.672
C00624=1191.476,123.787,-52.252,-178.556,6.120,148.673
C00625=1191.481,123.537,-52.232,-178.559,6.118,148.673
C00626=1191.487,123.288,-52.213,-178.562,6.118,148.674
C00627=1191.491,123.039,-52.193,-178.564,6.116,148.674
C00628=1191.496,122.790,-52.173,-178.567,6.114,148.675
C00629=1191.501,122.541,-52.153,-178.570,6.114,148.675
C00630=1191.506,122.292,-52.134,-178.572,6.112,148.676
C00631=1191.510,122.042,-52.115,-178.574,6.111,148.676
C00632=1191.515,121.793,-52.095,-178.578,6.110,148.677
C00633=1191.520,121.544,-52.076,-178.580,6.108,148.677
C00634=1191.524,121.295,-52.055,-178.582,6.107,148.678
C00635=1191.530,121.046,-52.036,-178.586,6.105,148.678
C00636=1191.534,120.796,-52.016,-178.588,6.105,148.679
C00637=1191.539,120.547,-51.997,-178.591,6.103,148.679
C00638=1191.544,120.298,-51.978,-178.594,6.101,148.680
C00639=1191.549,120.049,-51.958,-178.596,6.100,148.680
C00640=1191.553,119.799,-51.939,-178.599,6.099,148.681
C00641=1191.559,119.550,-51.919,-178.601,6.098,148.681
C00642=1191.563,119.301,-51.900,-178.604,6.096,148.681
C00643=1191.568,119.052,-51.881,-178.607,6.095,148.682
C00644=1191.573,118.803,-51.861,-178.609,6.094,148.682
C00645=1191.577,118.553,-51.842,-178.612,6.092,148.683
C00646=1191.583,118.304,-51.822,-178.614,6.092,148.683
C00647=1191.587,118.055,-51.803,-178.617,6.090,148.684
C00648=1191.592,117.806,-51.784,-178.619,6.089,148.684
C00649=1191.597,117.556,-51.764,-178.622,6.088,148.685
C00650=1191.602,117.307,-51.745,-178.625,6.086,148.685
C00651=1191.606,117.058,-51.726,-178.628,6.085,148.686
C00652=1191.611,116.809,-51.706,-178.630,6.084,148.686
C00653=1191.616,116.560,-51.687,-178.633,6.083,148.687
C00654=1191.620,116.311,-51.668,-178.636,6.081,148.687
C00655=1191.626,116.062,-51.649,-178.638,6.080,148.688
C00656=1191.630,115.812,-51.629,-178.641,6.078,148.688
C00657=1191.635,115.563,-51.609,-178.644,6.077,148.689
C00658=1191.640,115.314,-51.591,-178.646,6.076,148.689
C00659=1191.645,115.065,-51.571,-178.649,6.075,148.690
C00660=1191.650,114.816,-51.552,-178.651,6.074,148.690
C00661=1191.654,114.566,-51.533,-178.654,6.072,148.691
C00662=1191.660,114.317,-51.514,-178.657,6.072,148.691
C00663=1191.664,114.067,-51.494,-178.659,6.070,148.692
C00664=1191.669,113.819,-51.476,-178.661,6.069,148.692
C00665=1191.674,113.569,-51.456,-178.665,6.067,148.693
C00666=1191.679,113.320,-51.437,-178.667,6.066,148.693
C00667=1191.683,113.071,-51.418,-178.670,6.065,148.694
C00668=1191.689,112.822,-51.399,-178.673,6.063,148.694
C00669=1191.693,112.572,-51.380,-178.675,6.062,148.695
C00670=1191.698,112.324,-51.361,-178.678,6.061,148.695
C00671=1191.703,112.074,-51.341,-178.680,6.060,148.696
C00672=1191.708,111.825,-51.323,-178.683,6.059,148.696
C00673=1191.712,111.575,-51.304,-178.685,6.058,148.697
C00674=1191.717,111.327,-51.285,-178.688,6.056,148.697
C00675=1191.722,111.077,-51.265,-178.691,6.055,148.698
C00676=1191.727,110.828,-51.247,-178.693,6.054,148.698
C00677=1191.731,110.578,-51.228,-178.697,6.052,148.699
C00678=1191.737,110.329,-51.208,-178.699,6.051,148.699
C00679=1191.741,110.080,-51.189,-178.701,6.050,148.700
C00680=1191.746,109.831,-51.171,-178.704,6.049,148.700
C00681=1191.750,109.581,-51.152,-178.707,6.047,148.701
C00682=1191.756,109.333,-51.132,-178.709,6.047,148.701
C00683=1191.761,109.083,-51.114,-178.712,6.045,148.702
C00684=1191.765,108.834,-51.095,-178.715,6.044,148.702
C00685=1191.770,108.585,-51.076,-178.717,6.043,148.703
C00686=1191.775,108.335,-51.057,-178.719,6.042,148.703
C00687=1191.780,108.087,-51.038,-178.723,6.040,148.704
C00688=1191.785,107.836,-51.019,-178.725,6.039,148.704
C00689=1191.789,107.588,-51.001,-178.728,6.038,148.705
C00690=1191.795,107.339,-50.981,-178.730,6.037,148.705
C00691=1191.799,107.070,-50.962,-178.733,6.036,148.706
C00692=1191.805,106.802,-50.941,-178.736,6.034,148.706
C00693=1191.810,106.534,-50.922,-178.739,6.033,148.707
C00694=1191.815,106.265,-50.901,-178.742,6.032,148.708
C00695=1191.820,106.016,-50.882,-178.744,6.030,148.708
C00696=1191.825,105.766,-50.863,-178.747,6.029,148.708
C00697=1191.829,105.517,-50.845,-178.750,6.028,148.709
C00698=1191.835,105.268,-50.826,-178.752,6.027,148.709
C00699=1191.839,105.018,-50.807,-178.755,6.026,148.710
C00700=1191.844,104.769,-50.789,-178.757,6.025,148.710
C00701=1191.849,104.520,-50.770,-178.760,6.023,148.711
C00702=1191.853,104.271,-50.752,-178.763,6.022,148.712
C00703=1191.859,104.022,-50.732,-178.765,6.021,148.712
C00704=1191.864,103.773,-50.714,-178.768,6.020,148.713
C00705=1191.868,103.523,-50.695,-178.770,6.019,148.713
C00706=1191.873,103.274,-50.677,-178.773,6.018,148.714
C00707=1191.878,103.025,-50.658,-178.775,6.017,148.714
C00708=1191.882,102.775,-50.640,-178.779,6.015,148.715
C00709=1191.888,102.526,-50.621,-178.781,6.015,148.715
C00710=1191.892,102.277,-50.602,-178.784,6.013,148.716
C00711=1191.897,102.027,-50.584,-178.786,6.012,148.716
C00712=1191.902,101.779,-50.565,-178.789,6.011,148.717
C00713=1191.907,101.529,-50.547,-178.791,6.010,148.717
C00714=1191.911,101.279,-50.528,-178.794,6.008,148.718
C00715=1191.917,101.031,-50.509,-178.797,6.008,148.718
C00716=1191.922,100.781,-50.491,-178.799,6.006,148.719
C00717=1191.926,100.532,-50.473,-178.802,6.005,148.719
C00718=1191.931,100.283,-50.454,-178.805,6.004,148.720
C00719=1191.936,100.034,-50.435,-178.807,6.003,148.720
C00720=1191.941,99.784,-50.418,-178.810,6.001,148.721
C00721=1191.945,99.534,-50.399,-178.813,6.001,148.721
C00722=1191.951,99.286,-50.380,-178.815,5.999,148.722
C00723=1191.956,99.036,-50.362,-178.817,5.998,148.722
C00724=1191.961,98.787,-50.344,-178.820,5.997,148.723
C00725=1191.965,98.537,-50.326,-178.823,5.996,148.723
C00726=1191.970,98.289,-50.307,-178.825,5.995,148.724
C00727=1191.975,98.039,-50.288,-178.828,5.993,148.724
C00728=1191.980,97.790,-50.270,-178.831,5.993,148.725
C00729=1191.984,97.540,-50.252,-178.833,5.991,148.725
C00730=1191.989,97.292,-50.233,-178.836,5.991,148.726
C00731=1191.994,97.043,-50.215,-178.839,5.989,148.726
C00732=1192.000,96.793,-50.197,-178.841,5.988,148.727
C00733=1192.004,96.543,-50.178,-178.844,5.987,148.728
C00734=1192.009,96.294,-50.160,-178.847,5.986,148.728
C00735=1192.014,96.045,-50.142,-178.849,5.985,148.729
C00736=1192.018,95.796,-50.124,-178.852,5.984,148.729
C00737=1192.023,95.547,-50.106,-178.854,5.983,148.730
C00738=1192.028,95.297,-50.087,-178.857,5.981,148.730
C00739=1192.033,95.048,-50.069,-178.859,5.980,148.731
C00740=1192.038,94.799,-50.051,-178.863,5.979,148.731
C00741=1192.043,94.549,-50.033,-178.865,5.978,148.732
C00742=1192.048,94.300,-50.015,-178.867,5.978,148.732
C00743=1192.052,94.050,-49.997,-178.870,5.976,148.733
C00744=1192.057,93.801,-49.979,-178.873,5.975,148.733
C00745=1192.062,93.552,-49.961,-178.875,5.974,148.734
C00746=1192.068,93.302,-49.942,-178.878,5.973,148.735
C00747=1192.073,93.053,-49.924,-178.880,5.972,148.735
C00748=1192.078,92.804,-49.906,-178.883,5.971,148.736
C00749=1192.082,92.554,-49.888,-178.886,5.970,148.736
C00750=1192.087,92.305,-49.870,-178.889,5.968,148.737
C00751=1192.092,92.056,-49.852,-178.891,5.968,148.737
C00752=1192.097,91.807,-49.834,-178.894,5.966,148.738
C00753=1192.101,91.558,-49.816,-178.896,5.965,148.738
C00754=1192.106,91.308,-49.798,-178.899,5.965,148.739
C00755=1192.111,91.059,-49.780,-178.902,5.963,148.739
C00756=1192.116,90.809,-49.761,-178.904,5.962,148.740
C00757=1192.121,90.560,-49.743,-178.907,5.961,148.740
C00758=1192.125,90.311,-49.726,-178.910,5.960,148.741
C00759=1192.130,90.062,-49.708,-178.912,5.959,148.741
C00760=1192.135,89.813,-49.690,-178.915,5.958,148.742
C00761=1192.140,89.563,-49.672,-178.917,5.957,148.742
C00762=1192.145,89.314,-49.654,-178.920,5.955,148.743
C00763=1192.150,89.065,-49.636,-178.922,5.955,148.743
C00764=1192.155,88.816,-49.618,-178.925,5.954,148.744
C00765=1192.160,88.565,-49.600,-178.928,5.952,148.745
C00766=1192.164,88.316,-49.582,-178.930,5.952,148.745
C00767=1192.169,88.067,-49.564,-178.933,5.950,148.746
C00768=1192.174,87.818,-49.546,-178.936,5.949,148.746
C00769=1192.179,87.569,-49.528,-178.938,5.949,148.747
C00770=1192.184,87.320,-49.510,-178.941,5.947,148.747
C00771=1192.189,87.070,-49.493,-178.943,5.946,148.748
C00772=1192.193,86.821,-49.475,-178.946,5.945,148.748
C00773=1192.198,86.572,-49.457,-178.948,5.944,148.749
C00774=1192.203,86.323,-49.439,-178.951,5.943,148.750
C00775=1192.209,86.073,-49.422,-178.954,5.942,148.750
C00776=1192.213,85.824,-49.404,-178.956,5.941,148.751
C00777=1192.218,85.574,-49.386,-178.959,5.940,148.751
C00778=1192.223,85.325,-49.368,-178.962,5.939,148.752
C00779=1192.228,85.075,-49.351,-178.964,5.938,148.752
C00780=1192.233,84.826,-49.333,-178.967,5.937,148.753
C00781=1192.238,84.577,-49.316,-178.970,5.936,148.753
C00782=1192.242,84.328,-49.298,-178.972,5.935,148.754
C00783=1192.248,84.078,-49.280,-178.975,5.934,148.754
C00784=1192.253,83.829,-49.262,-178.977,5.933,148.755
C00785=1192.257,83.580,-49.244,-178.980,5.932,148.756
C00786=1192.263,83.330,-49.227,-178.983,5.931,148.756
C00787=1192.267,83.081,-49.210,-178.985,5.930,148.757
C00788=1192.272,82.832,-49.192,-178.987,5.929,148.757
C00789=1192.277,82.582,-49.175,-178.990,5.928,148.758
C00790=1192.282,82.333,-49.157,-178.993,5.927,148.758
C00791=1192.287,82.083,-49.139,-178.996,5.925,148.759
C00792=1192.291,81.835,-49.122,-178.998,5.925,148.759
C00793=1192.296,81.585,-49.104,-179.001,5.924,148.760
C00794=1192.301,81.336,-49.087,-179.004,5.923,148.760
C00795=1192.307,81.067,-49.067,-179.006,5.922,148.761
C00796=1192.312,80.798,-49.049,-179.009,5.920,148.762
C00797=1192.317,80.530,-49.029,-179.012,5.920,148.762
C00798=1192.322,80.262,-49.011,-179.015,5.918,148.763
C00799=1192.327,80.013,-48.993,-179.017,5.917,148.763
C00800=1192.332,79.763,-48.976,-179.020,5.917,148.764
C00801=1192.337,79.514,-48.958,-179.022,5.915,148.764
C00802=1192.342,79.265,-48.942,-179.025,5.915,148.765
C00803=1192.347,79.016,-48.924,-179.027,5.914,148.765
C00804=1192.352,78.766,-48.906,-179.030,5.912,148.766
C00805=1192.356,78.517,-48.889,-179.033,5.912,148.767
C00806=1192.361,78.267,-48.872,-179.035,5.911,148.767
C00807=1192.366,78.018,-48.854,-179.038,5.910,148.768
C00808=1192.371,77.768,-48.836,-179.041,5.909,148.768
C00809=1192.377,77.519,-48.820,-179.043,5.908,148.769
C00810=1192.381,77.270,-48.802,-179.046,5.906,148.769
C00811=1192.387,77.020,-48.785,-179.049,5.906,148.770
C00812=1192.391,76.772,-48.767,-179.051,5.905,148.770
C00813=1192.396,76.522,-48.750,-179.054,5.904,148.771
C00814=1192.401,76.273,-48.732,-179.056,5.903,148.772
C00815=1192.405,76.023,-48.716,-179.059,5.902,148.772
C00816=1192.411,75.773,-48.698,-179.062,5.901,148.773
C00817=1192.415,75.524,-48.681,-179.064,5.900,148.773
C00818=1192.421,75.275,-48.664,-179.067,5.899,148.774
C00819=1192.426,75.026,-48.647,-179.069,5.898,148.774
C00820=1192.430,74.777,-48.629,-179.072,5.897,148.775
C00821=1192.435,74.527,-48.612,-179.075,5.896,148.776
C00822=1192.440,74.277,-48.595,-179.077,5.896,148.776
C00823=1192.445,74.028,-48.577,-179.080,5.894,148.777
C00824=1192.450,73.778,-48.560,-179.082,5.893,148.777
C00825=1192.455,73.530,-48.544,-179.085,5.893,148.778
C00826=1192.460,73.280,-48.526,-179.088,5.891,148.778
C00827=1192.464,73.031,-48.509,-179.090,5.890,148.779
C00828=1192.470,72.781,-48.492,-179.093,5.890,148.780
C00829=1192.474,72.532,-48.475,-179.095,5.888,148.780
C00830=1192.480,72.283,-48.458,-179.098,5.888,148.781
C00831=1192.484,72.034,-48.441,-179.100,5.887,148.781
C00832=1192.489,71.784,-48.424,-179.103,5.886,148.782
C00833=1192.494,71.534,-48.406,-179.106,5.885,148.782
C00834=1192.499,71.285,-48.389,-179.108,5.884,148.783
C00835=1192.504,71.036,-48.372,-179.111,5.883,148.783
C00836=1192.509,70.787,-48.356,-179.113,5.882,148.784
C00837=1192.514,70.537,-48.338,-179.116,5.881,148.785
C00838=1192.519,70.287,-48.322,-179.119,5.881,148.785
C00839=1192.524,70.038,-48.304,-179.121,5.880,148.786
C00840=1192.529,69.789,-48.287,-179.124,5.878,148.786
C00841=1192.533,69.540,-48.271,-179.126,5.877,148.787
C00842=1192.538,69.290,-48.253,-179.129,5.877,148.787
C00843=1192.543,69.041,-48.237,-179.132,5.876,148.788
C00844=1192.549,68.792,-48.220,-179.134,5.875,148.788
C00845=1192.553,68.542,-48.203,-179.137,5.874,148.789
C00846=1192.558,68.293,-48.185,-179.139,5.873,148.790
C00847=1192.562,68.043,-48.169,-179.142,5.872,148.790
C00848=1192.568,67.794,-48.152,-179.145,5.871,148.791
C00849=1192.573,67.545,-48.135,-179.147,5.870,148.791
C00850=1192.577,67.295,-48.118,-179.150,5.870,148.792
C00851=1192.582,67.046,-48.101,-179.152,5.868,148.792
C00852=1192.588,66.797,-48.085,-179.155,5.868,148.793
C00853=1192.593,66.547,-48.067,-179.158,5.867,148.794
C00854=1192.597,66.298,-48.051,-179.160,5.865,148.794
C00855=1192.602,66.048,-48.034,-179.163,5.865,148.795
C00856=1192.608,65.799,-48.017,-179.166,5.864,148.795
C00857=1192.612,65.549,-48.001,-179.168,5.863,148.796
C00858=1192.617,65.300,-47.984,-179.171,5.862,148.797
C00859=1192.622,65.051,-47.967,-179.173,5.861,148.797
C00860=1192.627,64.801,-47.950,-179.176,5.861,148.798
C00861=1192.631,64.552,-47.934,-179.178,5.860,148.798
C00862=1192.637,64.303,-47.917,-179.181,5.858,148.799
C00863=1192.642,64.053,-47.900,-179.184,5.858,148.799
C00864=1192.646,63.804,-47.883,-179.186,5.857,148.800
C00865=1192.652,63.555,-47.866,-179.188,5.856,148.801
C00866=1192.656,63.305,-47.850,-179.192,5.855,148.801
C00867=1192.661,63.056,-47.833,-179.194,5.854,148.802
C00868=1192.667,62.807,-47.816,-179.196,5.854,148.802
C00869=1192.671,62.557,-47.800,-179.199,5.853,148.803
C00870=1192.676,62.307,-47.784,-179.201,5.852,148.803
C00871=1192.682,62.058,-47.767,-179.204,5.851,148.804
C00872=1192.686,61.809,-47.750,-179.207,5.850,148.805
C00873=1192.691,61.559,-47.733,-179.209,5.849,148.805
C00874=1192.696,61.310,-47.717,-179.212,5.849,148.806
C00875=1192.701,61.060,-47.700,-179.215,5.847,148.806
C00876=1192.706,60.811,-47.684,-179.217,5.847,148.807
C00877=1192.711,60.562,-47.668,-179.220,5.846,148.808
C00878=1192.715,60.312,-47.651,-179.222,5.845,148.808
C00879=1192.721,60.063,-47.634,-179.225,5.844,148.809
C00880=1192.726,59.814,-47.617,-179.228,5.843,148.809
C00881=1192.730,59.563,-47.601,-179.230,5.842,148.810
C00882=1192.736,59.315,-47.585,-179.233,5.842,148.810
C00883=1192.740,59.065,-47.568,-179.235,5.841,148.811
C00884=1192.746,58.816,-47.552,-179.238,5.840,148.812
C00885=1192.750,58.567,-47.535,-179.241,5.839,148.812
C00886=1192.756,58.317,-47.519,-179.243,5.838,148.813
C00887=1192.760,58.068,-47.503,-179.245,5.838,148.813
C00888=1192.765,57.818,-47.486,-179.249,5.836,148.814
C00889=1192.771,57.569,-47.470,-179.251,5.835,148.814
C00890=1192.775,57.319,-47.453,-179.253,5.835,148.815
C00891=1192.780,57.070,-47.437,-179.256,5.834,148.816
C00892=1192.785,56.821,-47.420,-179.258,5.833,148.816
C00893=1192.790,56.571,-47.404,-179.261,5.832,148.817
C00894=1192.795,56.322,-47.388,-179.264,5.832,148.818
C00895=1192.800,56.072,-47.371,-179.266,5.831,148.818
C00896=1192.805,55.823,-47.355,-179.269,5.830,148.819
C00897=1192.810,55.573,-47.338,-179.271,5.830,148.819
C00898=1192.815,55.324,-47.323,-179.274,5.828,148.820
C00899=1192.820,55.056,-47.305,-179.277,5.827,148.820
C00900=1192.825,54.787,-47.288,-179.279,5.827,148.821
C00901=1192.831,54.519,-47.270,-179.283,5.825,148.822
C00902=1192.836,54.250,-47.253,-179.285,5.825,148.822
C00903=1192.841,54.001,-47.236,-179.287,5.824,148.823
C00904=1192.847,53.751,-47.220,-179.290,5.824,148.823
C00905=1192.851,53.502,-47.203,-179.293,5.822,148.824
C00906=1192.857,53.252,-47.188,-179.295,5.821,148.825
C00907=1192.861,53.003,-47.171,-179.298,5.821,148.825
C00908=1192.867,52.753,-47.155,-179.301,5.820,148.826
C00909=1192.871,52.504,-47.139,-179.303,5.819,148.826
C00910=1192.876,52.255,-47.123,-179.306,5.818,148.827
C00911=1192.881,52.005,-47.107,-179.309,5.817,148.828
C00912=1192.886,51.756,-47.090,-179.311,5.817,148.828
C00913=1192.891,51.506,-47.074,-179.314,5.816,148.829
C00914=1192.896,51.257,-47.058,-179.316,5.816,148.829
C00915=1192.901,51.007,-47.042,-179.318,5.815,148.830
C00916=1192.906,50.759,-47.026,-179.322,5.813,148.831
C00917=1192.910,50.508,-47.010,-179.324,5.813,148.831
C00918=1192.916,50.259,-46.994,-179.326,5.812,148.832
C00919=1192.920,50.010,-46.978,-179.329,5.811,148.832
C00920=1192.926,49.760,-46.962,-179.332,5.811,148.833
C00921=1192.930,49.511,-46.945,-179.334,5.810,148.833
C00922=1192.936,49.261,-46.930,-179.337,5.809,148.834
C00923=1192.941,49.012,-46.913,-179.340,5.808,148.835
C00924=1192.945,48.762,-46.897,-179.342,5.807,148.835
C00925=1192.951,48.513,-46.882,-179.344,5.807,148.836
C00926=1192.955,48.263,-46.865,-179.347,5.806,148.837
C00927=1192.961,48.014,-46.850,-179.349,5.805,148.837
C00928=1192.964,47.765,-46.834,-179.352,5.804,148.838
C00929=1192.970,47.515,-46.818,-179.355,5.803,148.838
C00930=1192.975,47.266,-46.802,-179.357,5.803,148.839
C00931=1192.980,47.017,-46.786,-179.360,5.802,148.839
C00932=1192.985,46.767,-46.770,-179.362,5.801,148.840
C00933=1192.990,46.517,-46.754,-179.365,5.801,148.841
C00934=1192.995,46.268,-46.738,-179.367,5.800,148.841
C00935=1193.000,46.019,-46.722,-179.370,5.799,148.842
C00936=1193.005,45.769,-46.706,-179.373,5.798,148.842
C00937=1193.011,45.519,-46.691,-179.375,5.797,148.843
C00938=1193.015,45.271,-46.675,-179.378,5.797,148.844
C00939=1193.020,45.021,-46.659,-179.380,5.796,148.844
C00940=1193.025,44.771,-46.643,-179.383,5.795,148.845
C00941=1193.030,44.521,-46.627,-179.385,5.795,148.845
C00942=1193.035,44.273,-46.611,-179.389,5.794,148.846
C00943=1193.040,44.023,-46.596,-179.391,5.793,148.847
C00944=1193.044,43.773,-46.580,-179.393,5.792,148.847
C00945=1193.050,43.524,-46.565,-179.396,5.792,148.848
C00946=1193.055,43.275,-46.548,-179.398,5.791,148.848
C00947=1193.060,43.025,-46.532,-179.401,5.790,148.849
C00948=1193.065,42.776,-46.517,-179.403,5.790,148.850
C00949=1193.070,42.527,-46.502,-179.406,5.789,148.850
C00950=1193.074,42.276,-46.486,-179.409,5.787,148.851
C00951=1193.079,42.028,-46.470,-179.411,5.787,148.852
C00952=1193.085,41.778,-46.454,-179.414,5.786,148.852
C00953=1193.090,41.528,-46.438,-179.416,5.786,148.853
C00954=1193.094,41.279,-46.423,-179.419,5.785,148.853
C00955=1193.100,41.030,-46.407,-179.422,5.784,148.854
C00956=1193.105,40.780,-46.392,-179.424,5.784,148.854
C00957=1193.110,40.530,-46.376,-179.426,5.783,148.855
C00958=1193.115,40.281,-46.361,-179.430,5.782,148.856
C00959=1193.120,40.032,-46.345,-179.432,5.781,148.856
C00960=1193.124,39.782,-46.329,-179.434,5.780,148.857
C00961=1193.130,39.533,-46.313,-179.437,5.780,148.858
C00962=1193.134,39.284,-46.298,-179.439,5.779,148.858
C00963=1193.140,39.034,-46.282,-179.442,5.778,148.859
C00964=1193.145,38.784,-46.267,-179.444,5.778,148.859
C00965=1193.149,38.535,-46.252,-179.447,5.777,148.860
C00966=1193.155,38.286,-46.236,-179.449,5.777,148.860
C00967=1193.160,38.036,-46.220,-179.452,5.775,148.861
C00968=1193.165,37.786,-46.204,-179.455,5.775,148.862
C00969=1193.169,37.537,-46.189,-179.457,5.774,148.862
C00970=1193.175,37.288,-46.174,-179.460,5.773,148.863
C00971=1193.180,37.038,-46.158,-179.463,5.773,148.864
C00972=1193.184,36.788,-46.143,-179.465,5.772,148.864
C00973=1193.190,36.539,-46.127,-179.467,5.771,148.865
C00974=1193.195,36.290,-46.112,-179.470,5.771,148.865
C00975=1193.200,36.041,-46.097,-179.473,5.770,148.866
C00976=1193.204,35.790,-46.081,-179.475,5.769,148.867
C00977=1193.209,35.541,-46.066,-179.477,5.769,148.867
C00978=1193.215,35.292,-46.050,-179.481,5.768,148.868
C00979=1193.220,35.043,-46.035,-179.483,5.767,148.869
C00980=1193.225,34.793,-46.020,-179.485,5.766,148.869
C00981=1193.230,34.543,-46.004,-179.488,5.766,148.870
C00982=1193.234,34.294,-45.989,-179.491,5.765,148.870
C00983=1193.240,34.044,-45.974,-179.493,5.764,148.871
C00984=1193.245,33.795,-45.958,-179.496,5.764,148.871
C00985=1193.250,33.546,-45.943,-179.498,5.763,148.872
C00986=1193.255,33.296,-45.928,-179.501,5.763,148.873
C00987=1193.259,33.047,-45.912,-179.503,5.762,148.873
C00988=1193.265,32.797,-45.897,-179.506,5.761,148.874
C00989=1193.269,32.547,-45.882,-179.508,5.761,148.875
C00990=1193.275,32.298,-45.867,-179.511,5.759,148.875
C00991=1193.280,32.049,-45.851,-179.514,5.759,148.876
C00992=1193.285,31.800,-45.836,-179.516,5.758,148.876
C00993=1193.290,31.549,-45.820,-179.519,5.758,148.877
C00994=1193.295,31.300,-45.806,-179.521,5.757,148.878
C00995=1193.300,31.050,-45.790,-179.524,5.756,148.878
C00996=1193.305,30.801,-45.775,-179.526,5.756,148.879
C00997=1193.310,30.552,-45.760,-179.529,5.755,148.880
C00998=1193.315,30.302,-45.746,-179.531,5.754,148.880
C00999=1193.320,30.053,-45.730,-179.534,5.754,148.881
C01000=1193.324,29.803,-45.715,-179.536,5.753,148.881
C01001=1193.330,29.554,-45.699,-179.539,5.752,148.882
C01002=1193.335,29.304,-45.685,-179.541,5.752,148.883
C01003=1193.340,29.035,-45.668,-179.544,5.751,148.883
C01004=1193.346,28.767,-45.652,-179.547,5.750,148.884
C01005=1193.351,28.497,-45.636,-179.550,5.750,148.885
C01006=1193.356,28.229,-45.619,-179.552,5.749,148.885
C01007=1193.362,27.979,-45.604,-179.555,5.749,148.886
C01008=1193.367,27.730,-45.589,-179.557,5.748,148.886
C01009=1193.372,27.481,-45.574,-179.560,5.747,148.887
C01010=1193.377,27.231,-45.560,-179.562,5.747,148.888
C01011=1193.382,26.982,-45.545,-179.565,5.746,148.888
C01012=1193.387,26.733,-45.529,-179.567,5.745,148.889
C01013=1193.392,26.483,-45.515,-179.570,5.745,148.890
C01014=1193.397,26.233,-45.499,-179.573,5.744,148.890
C01015=1193.401,25.984,-45.484,-179.576,5.743,148.891
C01016=1193.406,25.734,-45.469,-179.578,5.742,148.891
C01017=1193.412,25.485,-45.454,-179.581,5.742,148.892
C01018=1193.417,25.235,-45.440,-179.583,5.741,148.893
C01019=1193.422,24.985,-45.424,-179.586,5.741,148.893
C01020=1193.427,24.736,-45.410,-179.588,5.740,148.894
C01021=1193.432,24.487,-45.395,-179.591,5.739,148.895
C01022=1193.437,24.237,-45.379,-179.593,5.739,148.895
C01023=1193.442,23.988,-45.365,-179.596,5.738,148.896
C01024=1193.447,23.738,-45.350,-179.598,5.737,148.896
C01025=1193.452,23.488,-45.335,-179.601,5.737,148.897
C01026=1193.457,23.239,-45.320,-179.603,5.736,148.898
C01027=1193.462,22.990,-45.306,-179.606,5.735,148.898
C01028=1193.467,22.740,-45.290,-179.608,5.735,148.899
C01029=1193.472,22.491,-45.276,-179.611,5.734,148.899
C01030=1193.477,22.241,-45.261,-179.614,5.734,148.900
C01031=1193.483,21.991,-45.246,-179.616,5.733,148.901
C01032=1193.487,21.742,-45.231,-179.618,5.733,148.901
C01033=1193.492,21.493,-45.217,-179.621,5.732,148.902
C01034=1193.497,21.244,-45.202,-179.624,5.732,148.903
C01035=1193.502,20.994,-45.187,-179.626,5.731,148.903
C01036=1193.507,20.744,-45.173,-179.628,5.730,148.904
C01037=1193.512,20.495,-45.158,-179.631,5.730,148.904
C01038=1193.517,20.245,-45.143,-179.634,5.729,148.905
C01039=1193.522,19.996,-45.128,-179.636,5.728,148.906
C01040=1193.527,19.746,-45.113,-179.639,5.728,148.906
C01041=1193.532,19.496,-45.099,-179.641,5.727,148.907
C01042=1193.537,19.247,-45.084,-179.644,5.727,148.908
C01043=1193.543,18.997,-45.069,-179.646,5.726,148.908
C01044=1193.547,18.748,-45.054,-179.649,5.725,148.909
C01045=1193.552,18.498,-45.040,-179.651,5.725,148.909
C01046=1193.557,18.249,-45.026,-179.654,5.724,148.910
C01047=1193.563,17.999,-45.010,-179.656,5.724,148.911
C01048=1193.568,17.749,-44.996,-179.659,5.723,148.911
C01049=1193.573,17.500,-44.982,-179.661,5.723,148.912
C01050=1193.578,17.251,-44.967,-179.664,5.722,148.913
C01051=1193.583,17.002,-44.953,-179.667,5.722,148.913
C01052=1193.588,16.752,-44.938,-179.669,5.721,148.914
C01053=1193.593,16.503,-44.923,-179.672,5.720,148.914
C01054=1193.598,16.253,-44.909,-179.674,5.720,148.915
C01055=1193.603,16.003,-44.894,-179.677,5.719,148.916
C01056=1193.608,15.753,-44.880,-179.679,5.718,148.916
C01057=1193.613,15.504,-44.865,-179.682,5.718,148.917
C01058=1193.618,15.255,-44.851,-179.684,5.717,148.918
C01059=1193.623,15.005,-44.836,-179.687,5.717,148.918
C01060=1193.628,14.755,-44.822,-179.689,5.716,148.919
C01061=1193.633,14.506,-44.807,-179.692,5.715,148.919
C01062=1193.638,14.257,-44.793,-179.694,5.715,148.920
C01063=1193.643,14.007,-44.778,-179.697,5.715,148.921
C01064=1193.648,13.757,-44.764,-179.699,5.714,148.921
C01065=1193.653,13.508,-44.750,-179.702,5.713,148.922
C01066=1193.658,13.259,-44.735,-179.705,5.713,148.923
C01067=1193.664,13.008,-44.720,-179.707,5.712,148.923
C01068=1193.669,12.759,-44.706,-179.709,5.711,148.924
C01069=1193.674,12.510,-44.692,-179.712,5.711,148.924
C01070=1193.679,12.260,-44.678,-179.715,5.710,148.925
C01071=1193.684,12.010,-44.663,-179.717,5.710,148.926
C01072=1193.689,11.761,-44.648,-179.720,5.709,148.927
C01073=1193.694,11.512,-44.634,-179.722,5.708,148.927
C01074=1193.699,11.262,-44.620,-179.725,5.708,148.928
C01075=1193.704,11.013,-44.606,-179.727,5.707,148.928
C01076=1193.709,10.763,-44.592,-179.730,5.707,148.929
C01077=1193.714,10.513,-44.577,-179.732,5.707,148.930
C01078=1193.719,10.264,-44.563,-179.734,5.706,148.930
C01079=1193.724,10.014,-44.549,-179.737,5.706,148.931
C01080=1193.729,9.764,-44.534,-179.740,5.705,148.932
C01081=1193.734,9.515,-44.521,-179.742,5.705,148.932
C01082=1193.739,9.266,-44.506,-179.744,5.704,148.933
C01083=1193.744,9.016,-44.492,-179.747,5.704,148.933
C01084=1193.749,8.767,-44.477,-179.750,5.703,148.934
C01085=1193.754,8.517,-44.463,-179.752,5.703,148.935
C01086=1193.760,8.268,-44.449,-179.755,5.702,148.935
C01087=1193.765,8.018,-44.434,-179.757,5.701,148.936
C01088=1193.769,7.769,-44.420,-179.760,5.701,148.937
C01089=1193.774,7.519,-44.406,-179.762,5.700,148.937
C01090=1193.780,7.270,-44.392,-179.765,5.699,148.938
C01091=1193.785,7.020,-44.378,-179.767,5.699,148.938
C01092=1193.790,6.770,-44.363,-179.770,5.698,148.939
C01093=1193.795,6.520,-44.350,-179.773,5.698,148.940
C01094=1193.800,6.270,-44.336,-179.775,5.697,148.940
C01095=1193.806,6.021,-44.322,-179.777,5.697,148.941
C01096=1193.811,5.772,-44.307,-179.779,5.697,148.942
C01097=1193.816,5.522,-44.293,-179.782,5.696,148.942
C01098=1193.820,5.273,-44.279,-179.785,5.696,148.943
C01099=1193.825,5.024,-44.266,-179.787,5.695,148.943
C01100=1193.830,4.774,-44.251,-179.790,5.695,148.944
C01101=1193.835,4.524,-44.237,-179.792,5.694,148.945
C01102=1193.841,4.275,-44.223,-179.795,5.694,148.946
C01103=1193.846,4.025,-44.209,-179.797,5.693,148.946
C01104=1193.851,3.776,-44.195,-179.800,5.692,148.947
C01105=1193.856,3.525,-44.181,-179.802,5.692,148.947
C01106=1193.861,3.277,-44.168,-179.805,5.691,148.948
C01107=1193.866,3.008,-44.152,-179.808,5.691,148.949
C01108=1193.871,2.739,-44.137,-179.810,5.690,148.949
C01109=1193.877,2.469,-44.122,-179.813,5.690,148.950
C01110=1193.882,2.200,-44.107,-179.816,5.689,148.951
C01111=1193.888,1.951,-44.093,-179.818,5.689,148.951
C01112=1193.893,1.701,-44.079,-179.820,5.688,148.952
C01113=1193.898,1.451,-44.065,-179.823,5.687,148.953
C01114=1193.904,1.202,-44.051,-179.826,5.687,148.953
C01115=1193.909,0.952,-44.037,-179.828,5.687,148.954
C01116=1193.913,0.703,-44.023,-179.831,5.686,148.954
C01117=1193.918,0.454,-44.009,-179.833,5.685,148.955
C01118=1193.924,0.203,-43.996,-179.835,5.685,148.956
C01119=1193.928,-0.047,-43.982,-179.838,5.685,148.957
C01120=1193.934,-0.296,-43.968,-179.841,5.685,148.957
C01121=1193.938,-0.545,-43.954,-179.843,5.684,148.958
C01122=1193.944,-0.795,-43.940,-179.845,5.683,148.958
C01123=1193.949,-1.044,-43.927,-179.848,5.683,148.959
C01124=1193.954,-1.294,-43.912,-179.851,5.682,148.960
C01125=1193.959,-1.544,-43.899,-179.853,5.682,148.960
C01126=1193.964,-1.793,-43.885,-179.856,5.681,148.961
C01127=1193.969,-2.043,-43.871,-179.858,5.680,148.962
C01128=1193.975,-2.292,-43.857,-179.860,5.681,148.962
C01129=1193.979,-2.542,-43.844,-179.863,5.680,148.963
C01130=1193.984,-2.791,-43.830,-179.865,5.679,148.963
C01131=1193.990,-3.040,-43.816,-179.868,5.679,148.964
C01132=1193.994,-3.290,-43.803,-179.870,5.678,148.965
C01133=1193.999,-3.540,-43.789,-179.873,5.678,148.965
C01134=1194.005,-3.790,-43.776,-179.876,5.677,148.966
C01135=1194.010,-4.040,-43.761,-179.878,5.677,148.967
C01136=1194.015,-4.288,-43.748,-179.881,5.676,148.967
C01137=1194.020,-4.539,-43.734,-179.883,5.676,148.968
C01138=1194.025,-4.788,-43.720,-179.885,5.676,148.969
C01139=1194.030,-5.038,-43.708,-179.888,5.675,148.969
C01140=1194.035,-5.287,-43.693,-179.890,5.675,148.970
C01141=1194.041,-5.536,-43.679,-179.893,5.674,148.971
C01142=1194.045,-5.786,-43.666,-179.895,5.674,148.971
C01143=1194.051,-6.035,-43.653,-179.898,5.673,148.972
C01144=1194.056,-6.286,-43.639,-179.901,5.673,148.973
C01145=1194.060,-6.535,-43.625,-179.903,5.672,148.973
C01146=1194.066,-6.785,-43.612,-179.905,5.672,148.974
C01147=1194.071,-7.034,-43.598,-179.908,5.672,148.974
C01148=1194.076,-7.284,-43.585,-179.910,5.671,148.975
C01149=1194.081,-7.533,-43.571,-179.912,5.670,148.976
C01150=1194.086,-7.783,-43.558,-179.915,5.670,148.976
C01151=1194.091,-8.032,-43.544,-179.918,5.669,148.977
C01152=1194.097,-8.282,-43.531,-179.920,5.669,148.978
C01153=1194.101,-8.532,-43.517,-179.923,5.668,148.978
C01154=1194.106,-8.782,-43.504,-179.925,5.668,148.979
C01155=1194.111,-9.031,-43.490,-179.927,5.668,148.980
C01156=1194.117,-9.281,-43.477,-179.930,5.667,148.980
C01157=1194.121,-9.530,-43.463,-179.933,5.667,148.981
C01158=1194.127,-9.780,-43.450,-179.935,5.666,148.982
C01159=1194.132,-10.029,-43.436,-179.937,5.666,148.982
C01160=1194.137,-10.279,-43.423,-179.940,5.665,148.983
C01161=1194.143,-10.529,-43.410,-179.942,5.665,148.983
C01162=1194.147,-10.778,-43.396,-179.945,5.665,148.984
C01163=1194.153,-11.028,-43.383,-179.948,5.665,148.985
C01164=1194.157,-11.277,-43.369,-179.950,5.664,148.985
C01165=1194.163,-11.527,-43.356,-179.952,5.663,148.986
C01166=1194.167,-11.777,-43.343,-179.955,5.663,148.987
C01167=1194.173,-12.026,-43.329,-179.958,5.662,148.987
C01168=1194.177,-12.276,-43.316,-179.960,5.663,148.988
C01169=1194.183,-12.525,-43.303,-179.962,5.662,148.989
C01170=1194.187,-12.775,-43.289,-179.965,5.661,148.989
C01171=1194.193,-13.024,-43.276,-179.967,5.661,148.990
C01172=1194.198,-13.274,-43.263,-179.970,5.660,148.991
C01173=1194.203,-13.523,-43.249,-179.973,5.660,148.991
C01174=1194.208,-13.773,-43.237,-179.975,5.659,148.992
C01175=1194.214,-14.023,-43.223,-179.977,5.659,148.992
C01176=1194.219,-14.272,-43.210,-179.979,5.659,148.993
C01177=1194.224,-14.522,-43.196,-179.982,5.658,148.994
C01178=1194.229,-14.771,-43.184,-179.984,5.658,148.994
C01179=1194.234,-15.021,-43.169,-179.987,5.657,148.995
C01180=1194.239,-15.270,-43.157,-179.990,5.657,148.996
C01181=1194.244,-15.520,-43.144,-179.992,5.657,148.996
C01182=1194.249,-15.770,-43.131,-179.994,5.656,148.997
C01183=1194.254,-16.019,-43.117,-179.996,5.656,148.998
C01184=1194.259,-16.269,-43.104,-179.999,5.655,148.998
C01185=1194.265,-16.518,-43.091,179.998,5.655,148.999
C01186=1194.270,-16.769,-43.078,179.996,5.654,149.000
C01187=1194.275,-17.018,-43.065,179.993,5.655,149.000
C01188=1194.280,-17.267,-43.052,179.991,5.654,149.001
C01189=1194.285,-17.517,-43.038,179.989,5.653,149.002
C01190=1194.290,-17.766,-43.025,179.986,5.653,149.002
C01191=1194.295,-18.017,-43.012,179.983,5.652,149.003
C01192=1194.301,-18.266,-42.999,179.981,5.652,149.004
C01193=1194.306,-18.515,-42.987,179.979,5.652,149.004
C01194=1194.311,-18.765,-42.972,179.976,5.651,149.005
C01195=1194.316,-19.014,-42.960,179.974,5.651,149.005
C01196=1194.320,-19.264,-42.947,179.971,5.650,149.006
C01197=1194.326,-19.514,-42.934,179.968,5.650,149.007
C01198=1194.331,-19.763,-42.921,179.966,5.649,149.007
C01199=1194.336,-20.013,-42.908,179.964,5.649,149.008
C01200=1194.342,-20.263,-42.895,179.962,5.649,149.009
C01201=1194.347,-20.512,-42.882,179.959,5.648,149.009
C01202=1194.351,-20.762,-42.869,179.956,5.648,149.010
C01203=1194.357,-21.011,-42.855,179.954,5.647,149.011
C01204=1194.362,-21.261,-42.843,179.952,5.647,149.011
C01205=1194.367,-21.511,-42.830,179.949,5.647,149.012
C01206=1194.372,-21.760,-42.817,179.947,5.647,149.013
C01207=1194.378,-22.010,-42.804,179.944,5.646,149.013
C01208=1194.382,-22.260,-42.791,179.942,5.645,149.014
C01209=1194.388,-22.509,-42.778,179.940,5.646,149.014
C01210=1194.393,-22.759,-42.765,179.937,5.645,149.015
C01211=1194.398,-23.028,-42.752,179.934,5.645,149.016
C01212=1194.404,-23.298,-42.737,179.932,5.644,149.017
C01213=1194.409,-23.567,-42.724,179.929,5.644,149.017
C01214=1194.415,-23.837,-42.710,179.926,5.643,149.018
C01215=1194.420,-24.087,-42.697,179.924,5.643,149.019
C01216=1194.425,-24.337,-42.684,179.921,5.642,149.019
C01217=1194.431,-24.586,-42.671,179.919,5.643,149.020
C01218=1194.436,-24.836,-42.658,179.917,5.642,149.021
C01219=1194.440,-25.086,-42.645,179.914,5.641,149.021
C01220=1194.445,-25.335,-42.633,179.912,5.641,149.022
C01221=1194.451,-25.584,-42.620,179.909,5.640,149.023
C01222=1194.456,-25.834,-42.607,179.907,5.641,149.023
C01223=1194.461,-26.084,-42.594,179.905,5.640,149.024
C01224=1194.466,-26.333,-42.581,179.902,5.639,149.024
C01225=1194.471,-26.583,-42.569,179.899,5.639,149.025
C01226=1194.476,-26.833,-42.556,179.897,5.639,149.026
C01227=1194.482,-27.082,-42.543,179.895,5.639,149.027
C01228=1194.487,-27.332,-42.531,179.892,5.638,149.027
C01229=1194.492,-27.581,-42.518,179.890,5.638,149.028
C01230=1194.497,-27.832,-42.505,179.887,5.637,149.028
C01231=1194.502,-28.081,-42.493,179.884,5.637,149.029
C01232=1194.507,-28.330,-42.480,179.883,5.637,149.030
C01233=1194.513,-28.580,-42.467,179.880,5.636,149.030
C01234=1194.517,-28.830,-42.454,179.878,5.636,149.031
C01235=1194.523,-29.080,-42.442,179.875,5.635,149.032
C01236=1194.528,-29.329,-42.429,179.873,5.636,149.032
C01237=1194.533,-29.578,-42.417,179.871,5.635,149.033
C01238=1194.537,-29.828,-42.404,179.868,5.634,149.034
C01239=1194.543,-30.078,-42.391,179.865,5.634,149.034
C01240=1194.548,-30.327,-42.379,179.863,5.633,149.035
C01241=1194.554,-30.577,-42.366,179.861,5.634,149.036
C01242=1194.559,-30.827,-42.353,179.858,5.633,149.036
C01243=1194.563,-31.077,-42.341,179.856,5.632,149.037
C01244=1194.569,-31.326,-42.328,179.853,5.632,149.038
C01245=1194.574,-31.576,-42.316,179.851,5.632,149.038
C01246=1194.579,-31.825,-42.303,179.848,5.632,149.039
C01247=1194.584,-32.074,-42.291,179.846,5.631,149.039
C01248=1194.589,-32.325,-42.278,179.843,5.631,149.040
C01249=1194.594,-32.574,-42.266,179.841,5.631,149.041
C01250=1194.599,-32.824,-42.253,179.839,5.630,149.041
C01251=1194.604,-33.073,-42.241,179.836,5.630,149.042
C01252=1194.610,-33.322,-42.228,179.834,5.629,149.043
C01253=1194.615,-33.572,-42.216,179.831,5.629,149.043
C01254=1194.620,-33.823,-42.203,179.829,5.629,149.044
C01255=1194.625,-34.072,-42.190,179.826,5.629,149.045
C01256=1194.631,-34.322,-42.178,179.824,5.628,149.045
C01257=1194.636,-34.571,-42.166,179.822,5.627,149.046
C01258=1194.641,-34.821,-42.153,179.820,5.628,149.047
C01259=1194.647,-35.070,-42.141,179.817,5.627,149.047
C01260=1194.652,-35.320,-42.129,179.814,5.627,149.048
C01261=1194.656,-35.570,-42.116,179.812,5.626,149.049
C01262=1194.662,-35.820,-42.104,179.810,5.626,149.049
C01263=1194.667,-36.069,-42.091,179.807,5.626,149.050
C01264=1194.672,-36.319,-42.079,179.805,5.625,149.051
C01265=1194.677,-36.568,-42.067,179.802,5.625,149.051
C01266=1194.682,-36.818,-42.054,179.800,5.625,149.052
C01267=1194.688,-37.068,-42.042,179.798,5.624,149.052
C01268=1194.693,-37.317,-42.030,179.795,5.624,149.053
C01269=1194.697,-37.567,-42.018,179.792,5.623,149.054
C01270=1194.702,-37.817,-42.005,179.790,5.624,149.055
C01271=1194.708,-38.066,-41.993,179.788,5.623,149.055
C01272=1194.713,-38.316,-41.981,179.786,5.622,149.056
C01273=1194.718,-38.565,-41.968,179.783,5.622,149.056
C01274=1194.723,-38.815,-41.956,179.781,5.622,149.057
C01275=1194.728,-39.064,-41.944,179.778,5.622,149.058
C01276=1194.734,-39.314,-41.932,179.775,5.621,149.059
C01277=1194.739,-39.564,-41.919,179.773,5.621,149.059
C01278=1194.744,-39.814,-41.907,179.771,5.621,149.060
C01279=1194.750,-40.063,-41.895,179.769,5.621,149.060
C01280=1194.755,-40.313,-41.883,179.766,5.620,149.061
C01281=1194.759,-40.563,-41.870,179.764,5.620,149.062
C01282=1194.764,-40.812,-41.859,179.762,5.620,149.062
C01283=1194.769,-41.062,-41.846,179.759,5.619,149.063
C01284=1194.775,-41.312,-41.834,179.756,5.619,149.064
C01285=1194.780,-41.561,-41.822,179.754,5.619,149.064
C01286=1194.785,-41.811,-41.810,179.752,5.619,149.065
C01287=1194.791,-42.061,-41.798,179.749,5.618,149.066
C01288=1194.796,-42.310,-41.785,179.747,5.617,149.066
C01289=1194.801,-42.560,-41.773,179.745,5.618,149.067
C01290=1194.806,-42.809,-41.761,179.742,5.617,149.068
C01291=1194.811,-43.059,-41.749,179.740,5.616,149.068
C01292=1194.816,-43.308,-41.737,179.738,5.617,149.069
C01293=1194.822,-43.558,-41.725,179.735,5.616,149.070
C01294=1194.827,-43.808,-41.713,179.732,5.616,149.070
C01295=1194.832,-44.058,-41.700,179.730,5.615,149.071
C01296=1194.837,-44.307,-41.689,179.728,5.615,149.071
C01297=1194.842,-44.557,-41.677,179.725,5.615,149.072
C01298=1194.847,-44.806,-41.665,179.723,5.614,149.073
C01299=1194.853,-45.056,-41.653,179.721,5.615,149.074
C01300=1194.858,-45.306,-41.640,179.718,5.614,149.074
C01301=1194.863,-45.555,-41.629,179.716,5.614,149.075
C01302=1194.868,-45.805,-41.617,179.713,5.613,149.075
C01303=1194.874,-46.055,-41.605,179.711,5.613,149.076
C01304=1194.879,-46.305,-41.592,179.708,5.613,149.077
C01305=1194.883,-46.554,-41.581,179.706,5.613,149.077
C01306=1194.889,-46.804,-41.569,179.704,5.613,149.078
C01307=1194.894,-47.053,-41.557,179.702,5.612,149.079
C01308=1194.899,-47.303,-41.545,179.699,5.612,149.079
C01309=1194.904,-47.553,-41.534,179.696,5.611,149.080
C01310=1194.909,-47.802,-41.521,179.695,5.611,149.081
C01311=1194.915,-48.052,-41.509,179.692,5.611,149.081
C01312=1194.920,-48.302,-41.497,179.689,5.610,149.082
C01313=1194.925,-48.552,-41.486,179.687,5.611,149.083
C01314=1194.930,-48.801,-41.473,179.685,5.610,149.083
C01315=1194.936,-49.071,-41.461,179.682,5.610,149.084
C01316=1194.941,-49.342,-41.448,179.679,5.609,149.085
C01317=1194.947,-49.612,-41.435,179.677,5.609,149.085
C01318=1194.953,-49.882,-41.423,179.674,5.609,149.086
C01319=1194.958,-50.132,-41.411,179.672,5.608,149.087
C01320=1194.963,-50.381,-41.398,179.670,5.608,149.087
C01321=1194.968,-50.631,-41.387,179.667,5.608,149.088
C01322=1194.973,-50.881,-41.375,179.665,5.608,149.089
C01323=1194.979,-51.131,-41.363,179.662,5.607,149.089
C01324=1194.983,-51.380,-41.352,179.660,5.607,149.090
C01325=1194.988,-51.629,-41.339,179.658,5.607,149.091
C01326=1194.994,-51.879,-41.328,179.655,5.607,149.091
C01327=1194.999,-52.129,-41.316,179.653,5.606,149.092
C01328=1195.005,-52.378,-41.305,179.651,5.606,149.093
C01329=1195.010,-52.628,-41.293,179.648,5.606,149.093
C01330=1195.015,-52.878,-41.282,179.646,5.605,149.094
C01331=1195.020,-53.128,-41.270,179.644,5.606,149.095
C01332=1195.025,-53.377,-41.258,179.641,5.605,149.095
C01333=1195.030,-53.627,-41.246,179.639,5.604,149.096
C01334=1195.035,-53.877,-41.234,179.637,5.605,149.096
C01335=1195.040,-54.126,-41.223,179.634,5.604,149.097
C01336=1195.046,-54.376,-41.211,179.631,5.604,149.098
C01337=1195.051,-54.625,-41.200,179.629,5.604,149.099
C01338=1195.056,-54.875,-41.188,179.627,5.603,149.099
C01339=1195.062,-55.125,-41.176,179.624,5.603,149.100
C01340=1195.066,-55.375,-41.165,179.622,5.602,149.101
C01341=1195.072,-55.625,-41.153,179.620,5.603,149.101
C01342=1195.077,-55.874,-41.142,179.617,5.602,149.102
C01343=1195.082,-56.124,-41.130,179.615,5.602,149.102
C01344=1195.087,-56.373,-41.119,179.613,5.602,149.103
C01345=1195.093,-56.623,-41.107,179.610,5.601,149.104
C01346=1195.097,-56.873,-41.096,179.607,5.601,149.104
C01347=1195.103,-57.123,-41.084,179.606,5.601,149.105
C01348=1195.108,-57.372,-41.072,179.603,5.601,149.106
C01349=1195.113,-57.622,-41.060,179.600,5.600,149.106
C01350=1195.118,-57.872,-41.049,179.598,5.600,149.107
C01351=1195.124,-58.121,-41.038,179.596,5.600,149.108
C01352=1195.129,-58.371,-41.026,179.594,5.599,149.108
C01353=1195.134,-58.621,-41.015,179.591,5.600,149.109
C01354=1195.139,-58.870,-41.003,179.589,5.599,149.110
C01355=1195.144,-59.120,-40.991,179.586,5.599,149.110
C01356=1195.150,-59.369,-40.980,179.585,5.599,149.111
C01357=1195.155,-59.619,-40.969,179.582,5.598,149.112
C01358=1195.160,-59.869,-40.957,179.579,5.598,149.112
C01359=1195.165,-60.119,-40.945,179.577,5.598,149.113
C01360=1195.169,-60.368,-40.934,179.575,5.597,149.113
C01361=1195.176,-60.618,-40.923,179.572,5.597,149.114
C01362=1195.180,-60.868,-40.912,179.570,5.597,149.115
C01363=1195.186,-61.118,-40.900,179.567,5.597,149.116
C01364=1195.191,-61.367,-40.889,179.565,5.597,149.116
C01365=1195.197,-61.616,-40.877,179.563,5.596,149.117
C01366=1195.201,-61.866,-40.866,179.561,5.596,149.117
C01367=1195.207,-62.116,-40.854,179.558,5.596,149.118
C01368=1195.211,-62.366,-40.843,179.556,5.596,149.119
C01369=1195.216,-62.616,-40.832,179.554,5.595,149.119
C01370=1195.222,-62.865,-40.821,179.552,5.595,149.120
C01371=1195.227,-63.115,-40.809,179.549,5.595,149.121
C01372=1195.233,-63.365,-40.798,179.546,5.595,149.121
C01373=1195.237,-63.614,-40.786,179.545,5.595,149.122
C01374=1195.244,-63.864,-40.775,179.542,5.594,149.123
C01375=1195.248,-64.114,-40.764,179.539,5.594,149.123
C01376=1195.253,-64.363,-40.753,179.537,5.594,149.124
C01377=1195.258,-64.613,-40.741,179.535,5.593,149.125
C01378=1195.264,-64.862,-40.730,179.532,5.593,149.125
C01379=1195.269,-65.112,-40.719,179.530,5.593,149.126
C01380=1195.274,-65.362,-40.708,179.528,5.593,149.127
C01381=1195.279,-65.611,-40.697,179.526,5.593,149.127
C01382=1195.285,-65.861,-40.685,179.523,5.592,149.128
C01383=1195.290,-66.112,-40.674,179.521,5.592,149.129
C01384=1195.295,-66.361,-40.663,179.519,5.592,149.129
C01385=1195.301,-66.610,-40.651,179.516,5.592,149.130
C01386=1195.305,-66.860,-40.640,179.514,5.591,149.130
C01387=1195.310,-67.110,-40.630,179.512,5.591,149.131
C01388=1195.316,-67.360,-40.618,179.509,5.591,149.132
C01389=1195.321,-67.609,-40.607,179.506,5.590,149.133
C01390=1195.326,-67.859,-40.596,179.505,5.590,149.133
C01391=1195.332,-68.109,-40.585,179.502,5.590,149.134
C01392=1195.337,-68.358,-40.573,179.500,5.590,149.134
C01393=1195.342,-68.608,-40.563,179.497,5.590,149.135
C01394=1195.348,-68.858,-40.551,179.495,5.589,149.136
C01395=1195.352,-69.107,-40.540,179.493,5.590,149.136
C01396=1195.357,-69.358,-40.529,179.490,5.589,149.137
C01397=1195.363,-69.607,-40.518,179.488,5.589,149.138
C01398=1195.368,-69.856,-40.507,179.486,5.589,149.138
C01399=1195.373,-70.107,-40.496,179.483,5.588,149.139
C01400=1195.378,-70.356,-40.485,179.481,5.589,149.140
C01401=1195.384,-70.606,-40.474,179.479,5.588,149.140
C01402=1195.389,-70.856,-40.463,179.476,5.587,149.141
C01403=1195.394,-71.105,-40.452,179.474,5.588,149.142
C01404=1195.399,-71.355,-40.441,179.472,5.587,149.142
C01405=1195.405,-71.604,-40.430,179.469,5.587,149.143
C01406=1195.410,-71.854,-40.419,179.467,5.587,149.143
C01407=1195.415,-72.104,-40.408,179.465,5.586,149.144
C01408=1195.420,-72.354,-40.398,179.463,5.587,149.145
C01409=1195.425,-72.603,-40.386,179.460,5.586,149.146
C01410=1195.431,-72.853,-40.374,179.458,5.586,149.146
C01411=1195.436,-73.103,-40.364,179.456,5.586,149.147
C01412=1195.441,-73.352,-40.353,179.453,5.586,149.147
C01413=1195.446,-73.602,-40.343,179.451,5.586,149.148
C01414=1195.452,-73.852,-40.331,179.449,5.585,149.149
C01415=1195.457,-74.102,-40.320,179.446,5.585,149.149
C01416=1195.462,-74.351,-40.309,179.444,5.585,149.150
C01417=1195.467,-74.601,-40.299,179.441,5.585,149.151
C01418=1195.472,-74.850,-40.288,179.439,5.584,149.151
C01419=1195.478,-75.122,-40.276,179.437,5.584,149.152
C01420=1195.484,-75.393,-40.264,179.434,5.584,149.153
C01421=1195.489,-75.663,-40.253,179.432,5.583,149.153
C01422=1195.495,-75.934,-40.240,179.430,5.584,149.154
C01423=1195.501,-76.183,-40.230,179.427,5.583,149.155
C01424=1195.505,-76.433,-40.219,179.424,5.583,149.155
C01425=1195.511,-76.683,-40.208,179.423,5.583,149.156
C01426=1195.517,-76.933,-40.198,179.420,5.582,149.157
C01427=1195.521,-77.183,-40.186,179.418,5.583,149.157
C01428=1195.527,-77.432,-40.176,179.415,5.582,149.158
C01429=1195.532,-77.682,-40.165,179.413,5.582,149.159
C01430=1195.537,-77.931,-40.155,179.411,5.582,149.159
C01431=1195.542,-78.181,-40.143,179.408,5.582,149.160
C01432=1195.548,-78.431,-40.132,179.406,5.582,149.161
C01433=1195.553,-78.681,-40.122,179.404,5.581,149.161
C01434=1195.559,-78.930,-40.111,179.401,5.581,149.162
C01435=1195.564,-79.180,-40.100,179.399,5.581,149.163
C01436=1195.569,-79.430,-40.090,179.397,5.581,149.163
C01437=1195.574,-79.679,-40.079,179.395,5.581,149.164
C01438=1195.579,-79.930,-40.068,179.392,5.580,149.165
C01439=1195.585,-80.179,-40.058,179.390,5.580,149.165
C01440=1195.589,-80.429,-40.047,179.388,5.580,149.166
C01441=1195.595,-80.678,-40.037,179.385,5.579,149.166
C01442=1195.600,-80.929,-40.026,179.383,5.580,149.167
C01443=1195.605,-81.177,-40.015,179.381,5.579,149.168
C01444=1195.610,-81.428,-40.005,179.379,5.579,149.168
C01445=1195.616,-81.677,-39.994,179.376,5.579,149.169
C01446=1195.620,-81.927,-39.983,179.374,5.578,149.170
C01447=1195.627,-82.177,-39.972,179.372,5.579,149.170
C01448=1195.632,-82.427,-39.962,179.370,5.578,149.171
C01449=1195.637,-82.677,-39.951,179.367,5.578,149.172
C01450=1195.642,-82.926,-39.940,179.365,5.578,149.172
C01451=1195.648,-83.176,-39.930,179.363,5.577,149.173
C01452=1195.653,-83.426,-39.919,179.361,5.578,149.174
C01453=1195.658,-83.675,-39.908,179.358,5.577,149.174
C01454=1195.663,-83.924,-39.898,179.356,5.578,149.175
C01455=1195.668,-84.175,-39.888,179.354,5.577,149.175
C01456=1195.674,-84.424,-39.877,179.351,5.576,149.176
C01457=1195.678,-84.674,-39.867,179.349,5.577,149.177
C01458=1195.684,-84.923,-39.857,179.347,5.576,149.177
C01459=1195.689,-85.173,-39.846,179.345,5.576,149.178
C01460=1195.694,-85.423,-39.836,179.342,5.576,149.179
C01461=1195.699,-85.673,-39.825,179.340,5.576,149.179
C01462=1195.705,-85.923,-39.815,179.338,5.575,149.180
C01463=1195.710,-86.172,-39.804,179.335,5.575,149.181
C01464=1195.715,-86.422,-39.793,179.333,5.575,149.181
C01465=1195.721,-86.671,-39.783,179.330,5.575,149.182
C01466=1195.726,-86.922,-39.773,179.329,5.575,149.183
C01467=1195.731,-87.171,-39.763,179.326,5.575,149.183
C01468=1195.736,-87.421,-39.752,179.324,5.575,149.184
C01469=1195.742,-87.670,-39.741,179.322,5.574,149.184
C01470=1195.747,-87.921,-39.730,179.319,5.574,149.185
C01471=1195.752,-88.170,-39.720,179.317,5.574,149.186
C01472=1195.758,-88.420,-39.710,179.315,5.573,149.186
C01473=1195.762,-88.670,-39.700,179.313,5.574,149.187
C01474=1195.768,-88.919,-39.690,179.310,5.573,149.188
C01475=1195.773,-89.169,-39.679,179.308,5.574,149.188
C01476=1195.778,-89.419,-39.669,179.306,5.573,149.189
C01477=1195.784,-89.668,-39.659,179.304,5.573,149.190
C01478=1195.789,-89.919,-39.648,179.301,5.573,149.190
C01479=1195.794,-90.168,-39.637,179.299,5.572,149.191
C01480=1195.800,-90.417,-39.627,179.297,5.572,149.192
C01481=1195.804,-90.667,-39.617,179.294,5.572,149.192
C01482=1195.810,-90.917,-39.607,179.292,5.572,149.193
C01483=1195.815,-91.167,-39.596,179.290,5.572,149.193
C01484=1195.820,-91.416,-39.586,179.288,5.572,149.194
C01485=1195.826,-91.666,-39.576,179.285,5.572,149.195
C01486=1195.831,-91.916,-39.565,179.283,5.571,149.195
C01487=1195.836,-92.166,-39.555,179.281,5.571,149.196
C01488=1195.841,-92.415,-39.546,179.278,5.571,149.197
C01489=1195.846,-92.665,-39.535,179.276,5.571,149.197
C01490=1195.852,-92.915,-39.525,179.274,5.570,149.198
C01491=1195.857,-93.164,-39.515,179.272,5.571,149.199
C01492=1195.862,-93.415,-39.504,179.269,5.570,149.199
C01493=1195.867,-93.664,-39.494,179.267,5.570,149.200
C01494=1195.873,-93.913,-39.484,179.265,5.570,149.201
C01495=1195.878,-94.164,-39.474,179.263,5.570,149.201
C01496=1195.883,-94.413,-39.463,179.260,5.569,149.202
C01497=1195.889,-94.663,-39.453,179.258,5.569,149.203
C01498=1195.894,-94.913,-39.444,179.256,5.569,149.203
C01499=1195.899,-95.163,-39.434,179.253,5.569,149.204
C01500=1195.905,-95.412,-39.423,179.251,5.569,149.204
C01501=1195.910,-95.663,-39.413,179.249,5.569,149.205
C01502=1195.915,-95.912,-39.403,179.247,5.569,149.206
C01503=1195.920,-96.161,-39.393,179.244,5.568,149.206
C01504=1195.925,-96.412,-39.383,179.242,5.569,149.207
C01505=1195.931,-96.661,-39.372,179.240,5.568,149.208
C01506=1195.936,-96.910,-39.363,179.238,5.568,149.208
C01507=1195.941,-97.160,-39.352,179.235,5.568,149.209
C01508=1195.947,-97.411,-39.343,179.233,5.567,149.209
C01509=1195.952,-97.660,-39.332,179.231,5.567,149.210
C01510=1195.957,-97.910,-39.323,179.228,5.567,149.211
C01511=1195.962,-98.160,-39.312,179.227,5.567,149.211
C01512=1195.968,-98.409,-39.302,179.224,5.567,149.212
C01513=1195.973,-98.659,-39.292,179.222,5.567,149.213
C01514=1195.978,-98.909,-39.283,179.220,5.566,149.213
C01515=1195.983,-99.159,-39.272,179.218,5.567,149.214
C01516=1195.989,-99.409,-39.262,179.215,5.566,149.215
C01517=1195.994,-99.658,-39.253,179.214,5.566,149.215
C01518=1196.000,-99.907,-39.242,179.211,5.566,149.216
C01519=1196.005,-100.158,-39.232,179.209,5.566,149.217
C01520=1196.010,-100.407,-39.223,179.207,5.565,149.217
C01521=1196.015,-100.657,-39.213,179.204,5.566,149.218
C01522=1196.021,-100.906,-39.202,179.202,5.565,149.219
C01523=1196.026,-101.178,-39.191,179.199,5.565,149.219
C01524=1196.032,-101.450,-39.181,179.197,5.565,149.220
C01525=1196.038,-101.721,-39.170,179.195,5.565,149.220
C01526=1196.044,-101.993,-39.160,179.192,5.564,149.221
C01527=1196.049,-102.243,-39.149,179.190,5.565,149.222
C01528=1196.053,-102.492,-39.140,179.187,5.564,149.223
C01529=1196.059,-102.742,-39.129,179.186,5.564,149.223
C01530=1196.065,-102.992,-39.120,179.183,5.564,149.224
C01531=1196.070,-103.241,-39.110,179.181,5.564,149.224
C01532=1196.075,-103.491,-39.100,179.179,5.563,149.225
C01533=1196.080,-103.741,-39.091,179.177,5.564,149.226
C01534=1196.086,-103.991,-39.081,179.174,5.563,149.226
C01535=1196.091,-104.240,-39.070,179.172,5.563,149.227
C01536=1196.096,-104.491,-39.061,179.170,5.563,149.228
C01537=1196.101,-104.740,-39.051,179.168,5.563,149.228
C01538=1196.106,-104.989,-39.041,179.166,5.562,149.229
C01539=1196.112,-105.240,-39.032,179.163,5.563,149.229
C01540=1196.117,-105.489,-39.022,179.161,5.562,149.230
C01541=1196.123,-105.738,-39.012,179.159,5.562,149.231
C01542=1196.128,-105.989,-39.002,179.156,5.562,149.231
C01543=1196.133,-106.238,-38.993,179.155,5.562,149.232
C01544=1196.138,-106.488,-38.982,179.152,5.562,149.233
C01545=1196.143,-106.738,-38.973,179.150,5.561,149.233
C01546=1196.149,-106.987,-38.963,179.148,5.561,149.234
C01547=1196.154,-107.237,-38.954,179.145,5.561,149.235
C01548=1196.159,-107.488,-38.944,179.143,5.561,149.235
C01549=1196.164,-107.737,-38.934,179.141,5.561,149.236
C01550=1196.170,-107.987,-38.925,179.139,5.561,149.236
C01551=1196.175,-108.236,-38.915,179.136,5.561,149.237
C01552=1196.181,-108.486,-38.906,179.135,5.561,149.238
C01553=1196.186,-108.736,-38.896,179.132,5.560,149.238
C01554=1196.191,-108.985,-38.886,179.130,5.561,149.239
C01555=1196.196,-109.236,-38.877,179.128,5.560,149.240
C01556=1196.201,-109.485,-38.866,179.126,5.560,149.240
C01557=1196.207,-109.735,-38.857,179.123,5.559,149.241
C01558=1196.212,-109.985,-38.847,179.121,5.560,149.241
C01559=1196.217,-110.234,-38.838,179.119,5.559,149.242
C01560=1196.223,-110.484,-38.828,179.117,5.559,149.243
C01561=1196.228,-110.734,-38.819,179.114,5.559,149.243
C01562=1196.234,-110.983,-38.809,179.112,5.559,149.244
C01563=1196.238,-111.234,-38.800,179.110,5.559,149.245
C01564=1196.244,-111.483,-38.790,179.108,5.559,149.245
C01565=1196.249,-111.733,-38.781,179.106,5.558,149.246
C01566=1196.255,-111.983,-38.770,179.104,5.559,149.246
C01567=1196.260,-112.233,-38.761,179.101,5.558,149.247
C01568=1196.265,-112.482,-38.751,179.099,5.558,149.248
C01569=1196.271,-112.732,-38.742,179.097,5.558,149.248
C01570=1196.275,-112.981,-38.733,179.095,5.558,149.249
C01571=1196.281,-113.231,-38.723,179.092,5.557,149.250
C01572=1196.286,-113.481,-38.714,179.090,5.558,149.250
C01573=1196.292,-113.731,-38.704,179.088,5.557,149.251
C01574=1196.297,-113.981,-38.695,179.086,5.557,149.252
C01575=1196.302,-114.231,-38.685,179.083,5.557,149.252
C01576=1196.307,-114.481,-38.676,179.082,5.557,149.253
C01577=1196.312,-114.730,-38.666,179.079,5.557,149.253
C01578=1196.318,-114.980,-38.657,179.078,5.557,149.254
C01579=1196.323,-115.230,-38.648,179.075,5.556,149.255
C01580=1196.328,-115.479,-38.638,179.073,5.557,149.255
C01581=1196.334,-115.729,-38.629,179.071,5.556,149.256
C01582=1196.339,-115.979,-38.620,179.069,5.556,149.257
C01583=1196.345,-116.229,-38.610,179.066,5.556,149.257
C01584=1196.350,-116.479,-38.601,179.064,5.556,149.258
C01585=1196.355,-116.728,-38.591,179.062,5.555,149.258
C01586=1196.361,-116.978,-38.582,179.060,5.555,149.259
C01587=1196.366,-117.228,-38.573,179.058,5.556,149.260
C01588=1196.371,-117.477,-38.563,179.055,5.555,149.260
C01589=1196.377,-117.727,-38.554,179.054,5.555,149.261
C01590=1196.382,-117.977,-38.545,179.051,5.555,149.262
C01591=1196.387,-118.226,-38.535,179.049,5.555,149.262
C01592=1196.393,-118.477,-38.526,179.047,5.555,149.263
C01593=1196.398,-118.726,-38.517,179.045,5.555,149.263
C01594=1196.403,-118.976,-38.508,179.042,5.554,149.264
C01595=1196.409,-119.226,-38.498,179.040,5.555,149.265
C01596=1196.414,-119.476,-38.489,179.038,5.554,149.265
C01597=1196.419,-119.726,-38.480,179.036,5.554,149.266
C01598=1196.425,-119.975,-38.470,179.034,5.554,149.266
C01599=1196.430,-120.225,-38.461,179.032,5.554,149.267
C01600=1196.435,-120.475,-38.452,179.029,5.554,149.268
C01601=1196.440,-120.725,-38.443,179.027,5.554,149.268
C01602=1196.446,-120.974,-38.433,179.025,5.553,149.269
C01603=1196.451,-121.224,-38.424,179.023,5.553,149.270
C01604=1196.456,-121.474,-38.415,179.020,5.553,149.270
C01605=1196.461,-121.724,-38.406,179.018,5.553,149.271
C01606=1196.467,-121.973,-38.396,179.016,5.552,149.271
C01607=1196.472,-122.223,-38.387,179.014,5.553,149.272
C01608=1196.477,-122.473,-38.378,179.012,5.552,149.273
C01609=1196.482,-122.723,-38.369,179.010,5.552,149.273
C01610=1196.488,-122.973,-38.360,179.008,5.552,149.274
C01611=1196.493,-123.222,-38.350,179.006,5.552,149.275
C01612=1196.498,-123.472,-38.341,179.003,5.552,149.275
C01613=1196.503,-123.722,-38.332,179.001,5.552,149.276
C01614=1196.509,-123.972,-38.323,178.999,5.552,149.276
C01615=1196.514,-124.222,-38.314,178.997,5.551,149.277
C01616=1196.520,-124.472,-38.305,178.995,5.552,149.278
C01617=1196.524,-124.721,-38.295,178.993,5.551,149.278
C01618=1196.530,-124.970,-38.287,178.991,5.551,149.279
C01619=1196.536,-125.220,-38.277,178.988,5.551,149.280
C01620=1196.541,-125.470,-38.268,178.986,5.551,149.280
C01621=1196.546,-125.720,-38.259,178.984,5.551,149.281
C01622=1196.552,-125.970,-38.251,178.982,5.551,149.281
C01623=1196.557,-126.220,-38.242,178.979,5.550,149.282
C01624=1196.563,-126.470,-38.232,178.978,5.550,149.282
C01625=1196.568,-126.719,-38.223,178.975,5.550,149.283
C01626=1196.573,-126.969,-38.214,178.974,5.550,149.284
C01627=1196.151,-126.980,-38.252,178.969,5.553,149.286
C01628=1196.146,-126.730,-38.261,178.972,5.554,149.285
C01629=1196.141,-126.480,-38.270,178.973,5.554,149.285
C01630=1196.135,-126.231,-38.280,178.975,5.553,149.284
C01631=1196.130,-125.981,-38.289,178.978,5.554,149.283
C01632=1196.125,-125.731,-38.298,178.980,5.554,149.283
C01633=1196.120,-125.481,-38.307,178.982,5.554,149.282
C01634=1196.115,-125.231,-38.316,178.984,5.554,149.281
C01635=1196.109,-124.981,-38.325,178.987,5.555,149.281
C01636=1196.103,-124.732,-38.334,178.988,5.555,149.280
C01637=1196.098,-124.482,-38.343,178.991,5.555,149.280
C01638=1196.093,-124.233,-38.353,178.993,5.555,149.279
C01639=1196.088,-123.983,-38.361,178.995,5.555,149.278
C01640=1196.082,-123.733,-38.371,178.997,5.555,149.278
C01641=1196.077,-123.483,-38.380,179.000,5.556,149.277
C01642=1196.072,-123.233,-38.389,179.002,5.555,149.276
C01643=1196.067,-122.983,-38.398,179.004,5.556,149.276
C01644=1196.061,-122.734,-38.408,179.006,5.556,149.275
C01645=1196.056,-122.484,-38.417,179.008,5.556,149.275
C01646=1196.051,-122.234,-38.426,179.010,5.556,149.274
C01647=1196.045,-121.984,-38.435,179.012,5.556,149.273
C01648=1196.040,-121.734,-38.444,179.014,5.556,149.273
C01649=1196.035,-121.485,-38.454,179.017,5.556,149.272
C01650=1196.030,-121.235,-38.463,179.019,5.557,149.272
C01651=1196.024,-120.985,-38.471,179.021,5.556,149.271
C01652=1196.018,-120.735,-38.481,179.023,5.557,149.270
C01653=1196.014,-120.486,-38.491,179.025,5.557,149.270
C01654=1196.008,-120.236,-38.499,179.028,5.557,149.269
C01655=1196.003,-119.986,-38.508,179.029,5.557,149.268
C01656=1195.997,-119.736,-38.518,179.032,5.558,149.268
C01657=1195.992,-119.487,-38.527,179.034,5.558,149.267
C01658=1195.987,-119.237,-38.536,179.036,5.558,149.267
C01659=1195.981,-118.987,-38.546,179.038,5.558,149.266
C01660=1195.977,-118.737,-38.555,179.041,5.558,149.265
C01661=1195.971,-118.488,-38.564,179.043,5.558,149.265
C01662=1195.965,-118.237,-38.574,179.045,5.559,149.264
C01663=1195.960,-117.988,-38.583,179.047,5.558,149.263
C01664=1195.955,-117.738,-38.592,179.050,5.559,149.263
C01665=1195.950,-117.488,-38.602,179.051,5.559,149.262
C01666=1195.944,-117.238,-38.611,179.054,5.559,149.262
C01667=1195.940,-116.989,-38.620,179.056,5.559,149.261
C01668=1195.934,-116.739,-38.630,179.058,5.559,149.260
C01669=1195.928,-116.489,-38.639,179.060,5.559,149.260
C01670=1195.924,-116.240,-38.648,179.063,5.560,149.259
C01671=1195.918,-115.990,-38.658,179.065,5.559,149.258
C01672=1195.913,-115.740,-38.667,179.067,5.560,149.258
C01673=1195.908,-115.491,-38.676,179.069,5.560,149.257
C01674=1195.902,-115.240,-38.686,179.072,5.560,149.256
C01675=1195.897,-114.991,-38.695,179.073,5.560,149.256
C01676=1195.891,-114.741,-38.705,179.076,5.561,149.255
C01677=1195.886,-114.491,-38.714,179.077,5.561,149.255
C01678=1195.881,-114.242,-38.723,179.080,5.560,149.254
C01679=1195.875,-113.992,-38.733,179.082,5.561,149.253
C01680=1195.870,-113.743,-38.743,179.084,5.561,149.253
C01681=1195.864,-113.492,-38.752,179.086,5.561,149.252
C01682=1195.860,-113.242,-38.762,179.088,5.561,149.252
C01683=1195.855,-112.993,-38.771,179.091,5.561,149.251
C01684=1195.849,-112.742,-38.780,179.093,5.561,149.250
C01685=1195.844,-112.493,-38.790,179.095,5.562,149.250
C01686=1195.838,-112.243,-38.800,179.097,5.561,149.249
C01687=1195.833,-111.994,-38.809,179.099,5.562,149.249
C01688=1195.827,-111.744,-38.819,179.101,5.562,149.248
C01689=1195.823,-111.494,-38.828,179.104,5.562,149.247
C01690=1195.817,-111.244,-38.838,179.106,5.562,149.247
C01691=1195.812,-110.995,-38.847,179.108,5.563,149.246
C01692=1195.806,-110.745,-38.857,179.110,5.562,149.245
C01693=1195.802,-110.495,-38.867,179.113,5.563,149.245
C01694=1195.796,-110.245,-38.876,179.115,5.562,149.244
C01695=1195.791,-109.996,-38.886,179.117,5.563,149.244
C01696=1195.786,-109.746,-38.895,179.119,5.563,149.243
C01697=1195.780,-109.496,-38.905,179.122,5.563,149.242
C01698=1195.775,-109.246,-38.914,179.124,5.564,149.242
C01699=1195.769,-108.997,-38.924,179.126,5.564,149.241
C01700=1195.765,-108.748,-38.934,179.129,5.564,149.240
C01701=1195.759,-108.497,-38.944,179.130,5.564,149.240
C01702=1195.754,-108.247,-38.953,179.133,5.564,149.239
C01703=1195.748,-107.997,-38.963,179.135,5.564,149.238
C01704=1195.744,-107.748,-38.972,179.137,5.565,149.238
C01705=1195.738,-107.498,-38.982,179.139,5.564,149.237
C01706=1195.732,-107.248,-38.992,179.141,5.565,149.237
C01707=1195.727,-106.999,-39.002,179.144,5.565,149.236
C01708=1195.722,-106.748,-39.012,179.146,5.565,149.235
C01709=1195.717,-106.499,-39.021,179.148,5.565,149.235
C01710=1195.711,-106.249,-39.031,179.150,5.566,149.234
C01711=1195.706,-106.000,-39.040,179.153,5.565,149.233
C01712=1195.701,-105.750,-39.050,179.155,5.566,149.233
C01713=1195.696,-105.500,-39.059,179.157,5.566,149.232
C01714=1195.691,-105.250,-39.070,179.160,5.566,149.231
C01715=1195.686,-105.001,-39.080,179.161,5.566,149.231
C01716=1195.680,-104.751,-39.089,179.164,5.566,149.230
C01717=1195.674,-104.501,-39.099,179.165,5.566,149.230
C01718=1195.669,-104.252,-39.109,179.168,5.567,149.229
C01719=1195.664,-104.001,-39.119,179.170,5.566,149.228
C01720=1195.659,-103.752,-39.128,179.172,5.567,149.228
C01721=1195.654,-103.502,-39.139,179.174,5.567,149.227
C01722=1195.648,-103.252,-39.148,179.177,5.567,149.226
C01723=1195.643,-103.003,-39.158,179.179,5.567,149.226
C01724=1195.638,-102.752,-39.168,179.181,5.568,149.225
C01725=1195.633,-102.503,-39.178,179.183,5.567,149.224
C01726=1195.627,-102.253,-39.187,179.186,5.568,149.224
C01727=1195.621,-102.004,-39.198,179.188,5.568,149.223
C01728=1195.616,-101.732,-39.208,179.190,5.568,149.223
C01729=1195.611,-101.460,-39.219,179.193,5.568,149.222
C01730=1195.605,-101.189,-39.230,179.195,5.568,149.221
C01731=1195.599,-100.918,-39.240,179.198,5.568,149.220
C01732=1195.594,-100.667,-39.251,179.200,5.569,149.220
C01733=1195.589,-100.418,-39.260,179.202,5.569,149.219
C01734=1195.583,-100.169,-39.270,179.205,5.569,149.218
C01735=1195.577,-99.918,-39.280,179.206,5.569,149.218
C01736=1195.573,-99.668,-39.290,179.209,5.570,149.217
C01737=1195.567,-99.419,-39.300,179.211,5.569,149.217
C01738=1195.562,-99.169,-39.310,179.213,5.570,149.216
C01739=1195.557,-98.920,-39.320,179.215,5.570,149.215
C01740=1195.552,-98.670,-39.331,179.218,5.570,149.215
C01741=1195.546,-98.420,-39.340,179.220,5.570,149.214
C01742=1195.541,-98.170,-39.350,179.222,5.571,149.213
C01743=1195.536,-97.921,-39.360,179.225,5.571,149.213
C01744=1195.531,-97.671,-39.370,179.227,5.571,149.212
C01745=1195.525,-97.421,-39.381,179.229,5.571,149.212
C01746=1195.520,-97.172,-39.390,179.231,5.571,149.211
C01747=1195.514,-96.922,-39.400,179.234,5.572,149.210
C01748=1195.509,-96.671,-39.410,179.236,5.571,149.210
C01749=1195.504,-96.422,-39.421,179.238,5.572,149.209
C01750=1195.499,-96.173,-39.430,179.240,5.572,149.208
C01751=1195.494,-95.922,-39.441,179.243,5.572,149.208
C01752=1195.488,-95.673,-39.451,179.245,5.572,149.207
C01753=1195.483,-95.423,-39.461,179.247,5.573,149.207
C01754=1195.478,-95.173,-39.471,179.249,5.572,149.206
C01755=1195.473,-94.924,-39.481,179.252,5.573,149.205
C01756=1195.467,-94.674,-39.492,179.254,5.573,149.205
C01757=1195.462,-94.425,-39.502,179.256,5.573,149.204
C01758=1195.456,-94.174,-39.512,179.259,5.573,149.203
C01759=1195.451,-93.925,-39.521,179.260,5.573,149.203
C01760=1195.446,-93.675,-39.531,179.263,5.574,149.202
C01761=1195.441,-93.425,-39.542,179.265,5.573,149.201
C01762=1195.435,-93.175,-39.552,179.268,5.574,149.201
C01763=1195.430,-92.926,-39.562,179.269,5.574,149.200
C01764=1195.425,-92.676,-39.572,179.272,5.574,149.199
C01765=1195.420,-92.426,-39.583,179.275,5.575,149.199
C01766=1195.415,-92.176,-39.593,179.276,5.575,149.198
C01767=1195.409,-91.927,-39.603,179.279,5.575,149.197
C01768=1195.404,-91.677,-39.614,179.281,5.575,149.197
C01769=1195.399,-91.427,-39.624,179.283,5.576,149.196
C01770=1195.394,-91.178,-39.634,179.285,5.575,149.196
C01771=1195.388,-90.928,-39.644,179.288,5.576,149.195
C01772=1195.383,-90.678,-39.655,179.290,5.576,149.194
C01773=1195.378,-90.428,-39.665,179.292,5.576,149.194
C01774=1195.372,-90.179,-39.675,179.295,5.576,149.193
C01775=1195.367,-89.929,-39.686,179.297,5.576,149.192
C01776=1195.362,-89.680,-39.697,179.299,5.577,149.192
C01777=1195.357,-89.430,-39.706,179.301,5.576,149.191
C01778=1195.352,-89.180,-39.717,179.304,5.577,149.190
C01779=1195.346,-88.930,-39.727,179.305,5.577,149.190
C01780=1195.341,-88.680,-39.737,179.308,5.577,149.189
C01781=1195.336,-88.431,-39.748,179.310,5.577,149.188
C01782=1195.331,-88.180,-39.758,179.312,5.578,149.188
C01783=1195.325,-87.931,-39.768,179.315,5.578,149.187
C01784=1195.319,-87.681,-39.779,179.317,5.578,149.187
C01785=1195.315,-87.432,-39.790,179.320,5.578,149.186
C01786=1195.310,-87.183,-39.800,179.321,5.578,149.185
C01787=1195.305,-86.932,-39.810,179.324,5.579,149.185
C01788=1195.299,-86.683,-39.820,179.326,5.578,149.184
C01789=1195.294,-86.432,-39.831,179.328,5.579,149.183
C01790=1195.289,-86.183,-39.841,179.331,5.579,149.183
C01791=1195.283,-85.933,-39.851,179.333,5.579,149.182
C01792=1195.278,-85.684,-39.863,179.336,5.579,149.181
C01793=1195.273,-85.434,-39.873,179.337,5.579,149.181
C01794=1195.268,-85.184,-39.883,179.340,5.580,149.180
C01795=1195.262,-84.934,-39.894,179.342,5.579,149.179
C01796=1195.257,-84.684,-39.904,179.344,5.580,149.179
C01797=1195.252,-84.435,-39.915,179.347,5.581,149.178
C01798=1195.247,-84.185,-39.926,179.349,5.580,149.178
C01799=1195.241,-83.935,-39.936,179.352,5.581,149.177
C01800=1195.236,-83.686,-39.946,179.353,5.581,149.176
C01801=1195.231,-83.436,-39.957,179.356,5.581,149.176
C01802=1195.225,-83.187,-39.968,179.359,5.582,149.175
C01803=1195.220,-82.937,-39.978,179.360,5.582,149.174
C01804=1195.215,-82.687,-39.988,179.363,5.582,149.174
C01805=1195.210,-82.437,-40.000,179.365,5.582,149.173
C01806=1195.205,-82.188,-40.010,179.368,5.582,149.172
C01807=1195.200,-81.938,-40.020,179.369,5.582,149.172
C01808=1195.194,-81.688,-40.031,179.372,5.582,149.171
C01809=1195.189,-81.438,-40.042,179.375,5.583,149.170
C01810=1195.184,-81.189,-40.052,179.376,5.583,149.170
C01811=1195.179,-80.939,-40.063,179.379,5.583,149.169
C01812=1195.173,-80.690,-40.074,179.381,5.583,149.168
C01813=1195.168,-80.439,-40.084,179.384,5.583,149.168
C01814=1195.163,-80.190,-40.094,179.386,5.584,149.167
C01815=1195.158,-79.940,-40.106,179.388,5.584,149.167
C01816=1195.152,-79.691,-40.116,179.391,5.584,149.166
C01817=1195.147,-79.440,-40.127,179.393,5.584,149.165
C01818=1195.142,-79.192,-40.137,179.395,5.585,149.165
C01819=1195.136,-78.941,-40.149,179.398,5.585,149.164
C01820=1195.131,-78.691,-40.159,179.400,5.585,149.163
C01821=1195.126,-78.442,-40.170,179.402,5.585,149.163
C01822=1195.121,-78.192,-40.181,179.404,5.585,149.162
C01823=1195.116,-77.943,-40.192,179.407,5.585,149.161
C01824=1195.111,-77.692,-40.202,179.409,5.586,149.161
C01825=1195.105,-77.443,-40.212,179.411,5.586,149.160
